LIN {X 0,Y 312.179,Z 630.649,A -85,B 0,C 180,E1 -16129.736,E2 -16129.736} C_VEL
LIN {X 0,Y 313.469,Z 619.934,A -85,B 0,C 180,E1 -16130.85,E2 -16130.85} C_VEL
LIN {X 0,Y 314.719,Z 608.145,A -85,B 0,C 180,E1 -16131.793,E2 -16131.793} C_VEL
LIN {X 0,Y 315.564,Z 595.146,A -85,B 0,C 180,E1 -16132.55,E2 -16132.55} C_VEL
LIN {X 0,Y 316.237,Z 582.572,A -85,B 0,C 180,E1 -16133.017,E2 -16133.017} C_VEL
LIN {X 0,Y 318.093,Z 505.284,A -85,B 0,C 180,E1 -16134.77,E2 -16134.77} C_VEL
LIN {X 0,Y 316.099,Z 493.068,A -85,B 0,C 180,E1 -16135.239,E2 -16135.239} C_VEL
LIN {X 0,Y 314.838,Z 489.465,A -85,B 0,C 180,E1 -16135.437,E2 -16135.437} C_VEL
LIN {X 0,Y 311.272,Z 484.306,A -85,B 0,C 180,E1 -16135.88,E2 -16135.88} C_VEL
LIN {X 0,Y 307.616,Z 479.185,A -85,B 0,C 180,E1 -16136.343,E2 -16136.343} C_VEL
LIN {X 0,Y 306.216,Z 475.627,A -85,B 0,C 180,E1 -16136.565,E2 -16136.565} C_VEL
LIN {X 0,Y 305.882,Z 473.673,A -85,B 0,C 180,E1 -16136.672,E2 -16136.672} C_VEL
LIN {X 0,Y 306.215,Z 468.394,A -85,B 0,C 180,E1 -16137.691,E2 -16137.691} C_VEL
LIN {X 0,Y 304.061,Z 457.591,A -85,B 0,C 180,E1 -16140.18,E2 -16140.18} C_VEL
LIN {X 0,Y 301.282,Z 446.622,A -85,B 0,C 180,E1 -16142.883,E2 -16142.883} C_VEL
LIN {X 0,Y 298.434,Z 436.313,A -85,B 0,C 180,E1 -16145.617,E2 -16145.617} C_VEL
LIN {X 0,Y 298.405,Z 436.31,A -85,B 0,C 180,E1 -16149.487,E2 -16149.487} C_VEL
LIN {X 0,Y 298.428,Z 436.305,A -85,B 0,C 180,E1 -16153.109,E2 -16153.109} C_VEL
LIN {X 0,Y 298.405,Z 436.311,A -85,B 0,C 180,E1 -16156.921,E2 -16156.921} C_VEL
LIN {X 0,Y 298.417,Z 436.315,A -85,B 0,C 180,E1 -16161.004,E2 -16161.004} C_VEL
LIN {X 0,Y 298.42,Z 436.293,A -85,B 0,C 180,E1 -16163.93,E2 -16163.93} C_VEL
LIN {X 0,Y 298.474,Z 436.324,A -85,B 0,C 180,E1 -16168.22,E2 -16168.22} C_VEL
LIN {X 0,Y 302.26,Z 454.228,A -85,B 0,C 180,E1 -16172.288,E2 -16172.288} C_VEL
LIN {X 0,Y 303.264,Z 459.72,A -85,B 0,C 180,E1 -16173.505,E2 -16173.505} C_VEL
LIN {X 0,Y 302.676,Z 470.14,A -85,B 0,C 180,E1 -16175.66,E2 -16175.66} C_VEL
LIN {X 0,Y 302.344,Z 474.693,A -85,B 0,C 180,E1 -16176.542,E2 -16176.542} C_VEL
LIN {X 0,Y 305.64,Z 502.289,A -85,B 0,C 180,E1 -16177.661,E2 -16177.661} C_VEL
LIN {X 0,Y 304.094,Z 552.285,A -85,B 0,C 180,E1 -16179.363,E2 -16179.363} C_VEL
LIN {X 0,Y 302.929,Z 586.5,A -85,B 0,C 180,E1 -16180.562,E2 -16180.562} C_VEL
LIN {X 0,Y 302.336,Z 599.637,A -85,B 0,C 180,E1 -16181.272,E2 -16181.272} C_VEL
LIN {X 0,Y 301.515,Z 612.031,A -85,B 0,C 180,E1 -16182.186,E2 -16182.186} C_VEL
LIN {X 0,Y 300.641,Z 624.863,A -85,B 0,C 180,E1 -16183.426,E2 -16183.426} C_VEL
LIN {X 0,Y 299.793,Z 636.649,A -85,B 0,C 180,E1 -16184.882,E2 -16184.882} C_VEL
LIN {X 0,Y 298.982,Z 646.67,A -85,B 0,C 180,E1 -16186.404,E2 -16186.404} C_VEL
LIN {X 0,Y 298.186,Z 655.778,A -85,B 0,C 180,E1 -16188.098,E2 -16188.098} C_VEL
LIN {X 0,Y 297.536,Z 664.71,A -85,B 0,C 180,E1 -16190.139,E2 -16190.139} C_VEL
LIN {X 0,Y 297.038,Z 671.83,A -85,B 0,C 180,E1 -16192.181,E2 -16192.181} C_VEL
LIN {X 0,Y 296.739,Z 677.24,A -85,B 0,C 180,E1 -16194.119,E2 -16194.119} C_VEL
LIN {X 0,Y 296.671,Z 681.217,A -85,B 0,C 180,E1 -16195.925,E2 -16195.925} C_VEL
LIN {X 0,Y 296.593,Z 683.617,A -85,B 0,C 180,E1 -16197.284,E2 -16197.284} C_VEL
LIN {X 0,Y 296.5,Z 685.517,A -85,B 0,C 180,E1 -16198.642,E2 -16198.642} C_VEL
LIN {X 0,Y 296.504,Z 686.947,A -85,B 0,C 180,E1 -16200,E2 -16200} C_VEL
LIN {X 0,Y 296.551,Z 687.964,A -85,B 0,C 180,E1 -16201.358,E2 -16201.358} C_VEL
LIN {X 0,Y 296.657,Z 688.505,A -85,B 0,C 180,E1 -16202.716,E2 -16202.716} C_VEL
LIN {X 0,Y 296.84,Z 688.612,A -85,B 0,C 180,E1 -16204.073,E2 -16204.073} C_VEL
LIN {X 0,Y 297.108,Z 688.306,A -85,B 0,C 180,E1 -16205.429,E2 -16205.429} C_VEL
LIN {X 0,Y 297.541,Z 687.205,A -85,B 0,C 180,E1 -16207.228,E2 -16207.228} C_VEL
LIN {X 0,Y 298.367,Z 684.756,A -85,B 0,C 180,E1 -16209.49,E2 -16209.49} C_VEL
LIN {X 0,Y 299.443,Z 681.451,A -85,B 0,C 180,E1 -16211.508,E2 -16211.508} C_VEL
LIN {X 0,Y 300.726,Z 677.059,A -85,B 0,C 180,E1 -16213.515,E2 -16213.515} C_VEL
LIN {X 0,Y 302.84,Z 670.363,A -85,B 0,C 180,E1 -16215.824,E2 -16215.824} C_VEL
LIN {X 0,Y 304.885,Z 663.119,A -85,B 0,C 180,E1 -16217.784,E2 -16217.784} C_VEL
LIN {X 0,Y 307.4,Z 654.112,A -85,B 0,C 180,E1 -16219.708,E2 -16219.708} C_VEL
LIN {X 0,Y 310.013,Z 643.808,A -85,B 0,C 180,E1 -16221.477,E2 -16221.477} C_VEL
LIN {X 0,Y 312.558,Z 632.651,A -85,B 0,C 180,E1 -16222.997,E2 -16222.997} C_VEL
LIN {X 0,Y 315.097,Z 619.91,A -85,B 0,C 180,E1 -16224.37,E2 -16224.37} C_VEL
LIN {X 0,Y 317.22,Z 607.363,A -85,B 0,C 180,E1 -16225.42,E2 -16225.42} C_VEL
LIN {X 0,Y 319.135,Z 593.779,A -85,B 0,C 180,E1 -16226.264,E2 -16226.264} C_VEL
LIN {X 0,Y 321.132,Z 574.897,A -85,B 0,C 180,E1 -16227.052,E2 -16227.052} C_VEL
LIN {X 0,Y 327.681,Z 513.253,A -85,B 0,C 180,E1 -16229.483,E2 -16229.483} C_VEL
LIN {X 0,Y 326.096,Z 500.284,A -85,B 0,C 180,E1 -16230.744,E2 -16230.744} C_VEL
LIN {X 0,Y 324.925,Z 493.87,A -85,B 0,C 180,E1 -16231.522,E2 -16231.522} C_VEL
LIN {X 0,Y 322.191,Z 487.566,A -85,B 0,C 180,E1 -16232.816,E2 -16232.816} C_VEL
LIN {X 0,Y 319.761,Z 482.587,A -85,B 0,C 180,E1 -16234.074,E2 -16234.074} C_VEL
LIN {X 0,Y 317.79,Z 478.528,A -85,B 0,C 180,E1 -16235.296,E2 -16235.296} C_VEL
LIN {X 0,Y 316.946,Z 473.742,A -85,B 0,C 180,E1 -16237.86,E2 -16237.86} C_VEL
LIN {X 0,Y 316.18,Z 470.661,A -85,B 0,C 180,E1 -16240.136,E2 -16240.136} C_VEL
LIN {X 0,Y 315.657,Z 468.393,A -85,B 0,C 180,E1 -16242.715,E2 -16242.715} C_VEL
LIN {X 0,Y 315.648,Z 467.284,A -85,B 0,C 180,E1 -16245.438,E2 -16245.438} C_VEL
LIN {X 0,Y 316.37,Z 467.578,A -85,B 0,C 180,E1 -16248.207,E2 -16248.207} C_VEL
LIN {X 0,Y 317.787,Z 469.248,A -85,B 0,C 180,E1 -16250.718,E2 -16250.718} C_VEL
LIN {X 0,Y 319.247,Z 471,A -85,B 0,C 180,E1 -16252.421,E2 -16252.421} C_VEL
LIN {X 0,Y 321.45,Z 475.13,A -85,B 0,C 180,E1 -16254.702,E2 -16254.702} C_VEL
LIN {X 0,Y 322.031,Z 482.327,A -85,B 0,C 180,E1 -16256.56,E2 -16256.56} C_VEL
LIN {X 0,Y 322.94,Z 486.125,A -85,B 0,C 180,E1 -16257.187,E2 -16257.187} C_VEL
LIN {X 0,Y 324.106,Z 499.658,A -85,B 0,C 180,E1 -16258.612,E2 -16258.612} C_VEL
LIN {X 0,Y 324.959,Z 512.771,A -85,B 0,C 180,E1 -16259.773,E2 -16259.773} C_VEL
LIN {X 0,Y 325.209,Z 525.188,A -85,B 0,C 180,E1 -16260.675,E2 -16260.675} C_VEL
LIN {X 0,Y 324.849,Z 536.213,A -85,B 0,C 180,E1 -16261.317,E2 -16261.317} C_VEL
LIN {X 0,Y 317.393,Z 605.626,A -85,B 0,C 180,E1 -16264.111,E2 -16264.111} C_VEL
LIN {X 0,Y 315.334,Z 619.995,A -85,B 0,C 180,E1 -16264.947,E2 -16264.947} C_VEL
LIN {X 0,Y 313.027,Z 633.136,A -85,B 0,C 180,E1 -16265.987,E2 -16265.987} C_VEL
LIN {X 0,Y 310.315,Z 646.166,A -85,B 0,C 180,E1 -16267.355,E2 -16267.355} C_VEL
LIN {X 0,Y 307.955,Z 656.683,A -85,B 0,C 180,E1 -16268.759,E2 -16268.759} C_VEL
LIN {X 0,Y 305.816,Z 665.619,A -85,B 0,C 180,E1 -16270.221,E2 -16270.221} C_VEL
LIN {X 0,Y 303.454,Z 674.922,A -85,B 0,C 180,E1 -16272.091,E2 -16272.091} C_VEL
LIN {X 0,Y 301.362,Z 682.883,A -85,B 0,C 180,E1 -16274.096,E2 -16274.096} C_VEL
LIN {X 0,Y 300.01,Z 688.24,A -85,B 0,C 180,E1 -16275.761,E2 -16275.761} C_VEL
LIN {X 0,Y 298.681,Z 693.437,A -85,B 0,C 180,E1 -16277.774,E2 -16277.774} C_VEL
LIN {X 0,Y 297.725,Z 697.491,A -85,B 0,C 180,E1 -16279.802,E2 -16279.802} C_VEL
LIN {X 0,Y 297.065,Z 700.459,A -85,B 0,C 180,E1 -16281.839,E2 -16281.839} C_VEL
LIN {X 0,Y 296.631,Z 702.706,A -85,B 0,C 180,E1 -16284.324,E2 -16284.324} C_VEL
LIN {X 0,Y 296.602,Z 703.351,A -85,B 0,C 180,E1 -16285.924,E2 -16285.924} C_VEL
LIN {X 0,Y 296.578,Z 703.936,A -85,B 0,C 180,E1 -16290,E2 -16290} C_VEL
LIN {X 0,Y 296.539,Z 703.71,A -85,B 0,C 180,E1 -16291.358,E2 -16291.358} C_VEL
LIN {X 0,Y 296.581,Z 703.091,A -85,B 0,C 180,E1 -16292.716,E2 -16292.716} C_VEL
LIN {X 0,Y 296.576,Z 702.079,A -85,B 0,C 180,E1 -16294.077,E2 -16294.077} C_VEL
LIN {X 0,Y 296.606,Z 700.394,A -85,B 0,C 180,E1 -16295.626,E2 -16295.626} C_VEL
LIN {X 0,Y 296.954,Z 696.415,A -85,B 0,C 180,E1 -16298.164,E2 -16298.164} C_VEL
LIN {X 0,Y 297.44,Z 691.994,A -85,B 0,C 180,E1 -16300.207,E2 -16300.207} C_VEL
LIN {X 0,Y 298.388,Z 685.265,A -85,B 0,C 180,E1 -16302.584,E2 -16302.584} C_VEL
LIN {X 0,Y 299.63,Z 677.919,A -85,B 0,C 180,E1 -16304.605,E2 -16304.605} C_VEL
LIN {X 0,Y 300.821,Z 670.414,A -85,B 0,C 180,E1 -16306.281,E2 -16306.281} C_VEL
LIN {X 0,Y 302.155,Z 661.31,A -85,B 0,C 180,E1 -16307.95,E2 -16307.95} C_VEL
LIN {X 0,Y 303.528,Z 652.857,A -85,B 0,C 180,E1 -16309.266,E2 -16309.266} C_VEL
LIN {X 0,Y 306.344,Z 641.93,A -85,B 0,C 180,E1 -16311.182,E2 -16311.182} C_VEL
LIN {X 0,Y 309.11,Z 630.854,A -85,B 0,C 180,E1 -16312.738,E2 -16312.738} C_VEL
LIN {X 0,Y 311.935,Z 618.673,A -85,B 0,C 180,E1 -16314.102,E2 -16314.102} C_VEL
LIN {X 0,Y 314.837,Z 605.198,A -85,B 0,C 180,E1 -16315.272,E2 -16315.272} C_VEL
LIN {X 0,Y 317.33,Z 591.028,A -85,B 0,C 180,E1 -16316.204,E2 -16316.204} C_VEL
LIN {X 0,Y 319.306,Z 576.399,A -85,B 0,C 180,E1 -16316.91,E2 -16316.91} C_VEL
LIN {X 0,Y 323.506,Z 532.518,A -85,B 0,C 180,E1 -16318.639,E2 -16318.639} C_VEL
LIN {X 0,Y 323.456,Z 521.067,A -85,B 0,C 180,E1 -16319.348,E2 -16319.348} C_VEL
LIN {X 0,Y 322.626,Z 507.921,A -85,B 0,C 180,E1 -16320.374,E2 -16320.374} C_VEL
LIN {X 0,Y 321.365,Z 496.387,A -85,B 0,C 180,E1 -16321.471,E2 -16321.471} C_VEL
LIN {X 0,Y 319.999,Z 486.16,A -85,B 0,C 180,E1 -16322.596,E2 -16322.596} C_VEL
LIN {X 0,Y 317.791,Z 480.722,A -85,B 0,C 180,E1 -16323.689,E2 -16323.689} C_VEL
LIN {X 0,Y 314.86,Z 474.071,A -85,B 0,C 180,E1 -16325.29,E2 -16325.29} C_VEL
LIN {X 0,Y 310.76,Z 465.64,A -85,B 0,C 180,E1 -16328.018,E2 -16328.018} C_VEL
LIN {X 0,Y 307.898,Z 460.525,A -85,B 0,C 180,E1 -16330.617,E2 -16330.617} C_VEL
LIN {X 0,Y 306.358,Z 457.152,A -85,B 0,C 180,E1 -16333.019,E2 -16333.019} C_VEL
LIN {X 0,Y 305.84,Z 455.139,A -85,B 0,C 180,E1 -16335.427,E2 -16335.427} C_VEL
LIN {X 0,Y 306.109,Z 454.482,A -85,B 0,C 180,E1 -16337.282,E2 -16337.282} C_VEL
LIN {X 0,Y 307.974,Z 454.466,A -85,B 0,C 180,E1 -16340.285,E2 -16340.285} C_VEL
LIN {X 0,Y 310.912,Z 457.042,A -85,B 0,C 180,E1 -16343.023,E2 -16343.023} C_VEL
LIN {X 0,Y 311.867,Z 458.038,A -85,B 0,C 180,E1 -16343.717,E2 -16343.717} C_VEL
LIN {X 0,Y 315.045,Z 461.304,A -85,B 0,C 180,E1 -16345.629,E2 -16345.629} C_VEL
LIN {X 0,Y 318.095,Z 465.04,A -85,B 0,C 180,E1 -16347.173,E2 -16347.173} C_VEL
LIN {X 0,Y 321.283,Z 469.175,A -85,B 0,C 180,E1 -16348.553,E2 -16348.553} C_VEL
LIN {X 0,Y 325.804,Z 475.942,A -85,B 0,C 180,E1 -16350.309,E2 -16350.309} C_VEL
LIN {X 0,Y 327.91,Z 479.942,A -85,B 0,C 180,E1 -16351.098,E2 -16351.098} C_VEL
LIN {X 0,Y 321.93,Z 534.652,A -85,B 0,C 180,E1 -16353.283,E2 -16353.283} C_VEL
LIN {X 0,Y 320.518,Z 549.088,A -85,B 0,C 180,E1 -16354.028,E2 -16354.028} C_VEL
LIN {X 0,Y 319.036,Z 561.414,A -85,B 0,C 180,E1 -16354.908,E2 -16354.908} C_VEL
LIN {X 0,Y 316.909,Z 574.47,A -85,B 0,C 180,E1 -16356.124,E2 -16356.124} C_VEL
LIN {X 0,Y 314.538,Z 586.079,A -85,B 0,C 180,E1 -16357.503,E2 -16357.503} C_VEL
LIN {X 0,Y 312.356,Z 595.61,A -85,B 0,C 180,E1 -16358.9,E2 -16358.9} C_VEL
LIN {X 0,Y 310.19,Z 604.328,A -85,B 0,C 180,E1 -16360.477,E2 -16360.477} C_VEL
LIN {X 0,Y 308.126,Z 611.561,A -85,B 0,C 180,E1 -16362.066,E2 -16362.066} C_VEL
LIN {X 0,Y 305.926,Z 618.701,A -85,B 0,C 180,E1 -16363.998,E2 -16363.998} C_VEL
LIN {X 0,Y 303.95,Z 624.421,A -85,B 0,C 180,E1 -16365.949,E2 -16365.949} C_VEL
LIN {X 0,Y 302.306,Z 628.869,A -85,B 0,C 180,E1 -16367.923,E2 -16367.923} C_VEL
LIN {X 0,Y 301.275,Z 631.244,A -85,B 0,C 180,E1 -16369.244,E2 -16369.244} C_VEL
LIN {X 0,Y 300.367,Z 633.147,A -85,B 0,C 180,E1 -16370.573,E2 -16370.573} C_VEL
LIN {X 0,Y 299.648,Z 634.568,A -85,B 0,C 180,E1 -16371.91,E2 -16371.91} C_VEL
LIN {X 0,Y 299.074,Z 635.563,A -85,B 0,C 180,E1 -16373.252,E2 -16373.252} C_VEL
LIN {X 0,Y 298.54,Z 636.139,A -85,B 0,C 180,E1 -16374.597,E2 -16374.597} C_VEL
LIN {X 0,Y 298.063,Z 636.261,A -85,B 0,C 180,E1 -16375.944,E2 -16375.944} C_VEL
LIN {X 0,Y 297.707,Z 635.969,A -85,B 0,C 180,E1 -16377.294,E2 -16377.294} C_VEL
LIN {X 0,Y 297.453,Z 635.269,A -85,B 0,C 180,E1 -16378.646,E2 -16378.646} C_VEL
LIN {X 0,Y 297.297,Z 634.103,A -85,B 0,C 180,E1 -16380,E2 -16380} C_VEL
LIN {X 0,Y 297.313,Z 631.537,A -85,B 0,C 180,E1 -16382.032,E2 -16382.032} C_VEL
LIN {X 0,Y 297.458,Z 627.933,A -85,B 0,C 180,E1 -16384.065,E2 -16384.065} C_VEL
LIN {X 0,Y 297.67,Z 623.195,A -85,B 0,C 180,E1 -16386.099,E2 -16386.099} C_VEL
LIN {X 0,Y 298.012,Z 616.074,A -85,B 0,C 180,E1 -16388.476,E2 -16388.476} C_VEL
LIN {X 0,Y 298.523,Z 608.297,A -85,B 0,C 180,E1 -16390.513,E2 -16390.513} C_VEL
LIN {X 0,Y 299.307,Z 598.647,A -85,B 0,C 180,E1 -16392.545,E2 -16392.545} C_VEL
LIN {X 0,Y 300.184,Z 587.588,A -85,B 0,C 180,E1 -16394.404,E2 -16394.404} C_VEL
LIN {X 0,Y 300.941,Z 576.409,A -85,B 0,C 180,E1 -16395.927,E2 -16395.927} C_VEL
LIN {X 0,Y 301.806,Z 564.264,A -85,B 0,C 180,E1 -16397.239,E2 -16397.239} C_VEL
LIN {X 0,Y 302.449,Z 550.933,A -85,B 0,C 180,E1 -16398.37,E2 -16398.37} C_VEL
LIN {X 0,Y 303.109,Z 536.628,A -85,B 0,C 180,E1 -16399.25,E2 -16399.25} C_VEL
LIN {X 0,Y 303.479,Z 522.328,A -85,B 0,C 180,E1 -16399.841,E2 -16399.841} C_VEL
LIN {X 0,Y 305.469,Z 458.71,A -85,B 0,C 180,E1 -16402.009,E2 -16402.009} C_VEL
LIN {X 0,Y 298.462,Z 436.299,A -85,B 0,C 180,E1 -16403.13,E2 -16403.13} C_VEL
LIN {X 0,Y 298.486,Z 436.303,A -85,B 0,C 180,E1 -16406.575,E2 -16406.575} C_VEL
LIN {X 0,Y 298.419,Z 436.314,A -85,B 0,C 180,E1 -16409.641,E2 -16409.641} C_VEL
LIN {X 0,Y 298.397,Z 436.29,A -85,B 0,C 180,E1 -16412.8,E2 -16412.8} C_VEL
LIN {X 0,Y 298.449,Z 436.311,A -85,B 0,C 180,E1 -16416.808,E2 -16416.808} C_VEL
LIN {X 0,Y 298.411,Z 436.3,A -85,B 0,C 180,E1 -16419.486,E2 -16419.486} C_VEL
LIN {X 0,Y 298.4,Z 436.321,A -85,B 0,C 180,E1 -16423.103,E2 -16423.103} C_VEL
LIN {X 0,Y 298.405,Z 436.305,A -85,B 0,C 180,E1 -16426.921,E2 -16426.921} C_VEL
LIN {X 0,Y 298.417,Z 436.309,A -85,B 0,C 180,E1 -16431.004,E2 -16431.004} C_VEL
LIN {X 0,Y 298.429,Z 436.362,A -85,B 0,C 180,E1 -16434.547,E2 -16434.547} C_VEL
LIN {X 0,Y 301.7,Z 448.047,A -85,B 0,C 180,E1 -16437.603,E2 -16437.603} C_VEL
LIN {X 0,Y 304.671,Z 460.525,A -85,B 0,C 180,E1 -16440.647,E2 -16440.647} C_VEL
LIN {X 0,Y 306.128,Z 467.823,A -85,B 0,C 180,E1 -16442.314,E2 -16442.314} C_VEL
LIN {X 0,Y 305.847,Z 473.764,A -85,B 0,C 180,E1 -16443.462,E2 -16443.462} C_VEL
LIN {X 0,Y 310.58,Z 499.528,A -85,B 0,C 180,E1 -16444.558,E2 -16444.558} C_VEL
LIN {X 0,Y 311.587,Z 506.235,A -85,B 0,C 180,E1 -16444.814,E2 -16444.814} C_VEL
LIN {X 0,Y 309.769,Z 580.357,A -85,B 0,C 180,E1 -16446.518,E2 -16446.518} C_VEL
LIN {X 0,Y 309.181,Z 593.095,A -85,B 0,C 180,E1 -16446.958,E2 -16446.958} C_VEL
LIN {X 0,Y 308.244,Z 605.504,A -85,B 0,C 180,E1 -16447.637,E2 -16447.637} C_VEL
LIN {X 0,Y 307.165,Z 617.161,A -85,B 0,C 180,E1 -16448.526,E2 -16448.526} C_VEL
LIN {X 0,Y 305.785,Z 628.549,A -85,B 0,C 180,E1 -16449.658,E2 -16449.658} C_VEL
LIN {X 0,Y 304.37,Z 638.81,A -85,B 0,C 180,E1 -16450.965,E2 -16450.965} C_VEL
LIN {X 0,Y 303.085,Z 648.214,A -85,B 0,C 180,E1 -16452.455,E2 -16452.455} C_VEL
LIN {X 0,Y 301.533,Z 656.811,A -85,B 0,C 180,E1 -16454.106,E2 -16454.106} C_VEL
LIN {X 0,Y 300.238,Z 663.905,A -85,B 0,C 180,E1 -16455.772,E2 -16455.772} C_VEL
LIN {X 0,Y 299.08,Z 670.867,A -85,B 0,C 180,E1 -16457.79,E2 -16457.79} C_VEL
LIN {X 0,Y 298.096,Z 676.399,A -85,B 0,C 180,E1 -16459.815,E2 -16459.815} C_VEL
LIN {X 0,Y 297.441,Z 680.736,A -85,B 0,C 180,E1 -16461.85,E2 -16461.85} C_VEL
LIN {X 0,Y 297.107,Z 683.412,A -85,B 0,C 180,E1 -16463.467,E2 -16463.467} C_VEL
LIN {X 0,Y 296.766,Z 686.296,A -85,B 0,C 180,E1 -16465.926,E2 -16465.926} C_VEL
LIN {X 0,Y 296.53,Z 687.905,A -85,B 0,C 180,E1 -16468.642,E2 -16468.642} C_VEL
LIN {X 0,Y 296.512,Z 688.138,A -85,B 0,C 180,E1 -16470,E2 -16470} C_VEL
LIN {X 0,Y 296.53,Z 687.944,A -85,B 0,C 180,E1 -16471.358,E2 -16471.358} C_VEL
LIN {X 0,Y 296.765,Z 686.385,A -85,B 0,C 180,E1 -16474.074,E2 -16474.074} C_VEL
LIN {X 0,Y 297.076,Z 683.66,A -85,B 0,C 180,E1 -16476.482,E2 -16476.482} C_VEL
LIN {X 0,Y 297.608,Z 679.632,A -85,B 0,C 180,E1 -16478.83,E2 -16478.83} C_VEL
LIN {X 0,Y 298.379,Z 674.966,A -85,B 0,C 180,E1 -16480.861,E2 -16480.861} C_VEL
LIN {X 0,Y 299.636,Z 667.955,A -85,B 0,C 180,E1 -16483.22,E2 -16483.22} C_VEL
LIN {X 0,Y 300.963,Z 660.269,A -85,B 0,C 180,E1 -16485.231,E2 -16485.231} C_VEL
LIN {X 0,Y 302.672,Z 650.694,A -85,B 0,C 180,E1 -16487.221,E2 -16487.221} C_VEL
LIN {X 0,Y 304.1,Z 640.694,A -85,B 0,C 180,E1 -16488.878,E2 -16488.878} C_VEL
LIN {X 0,Y 305.753,Z 629.442,A -85,B 0,C 180,E1 -16490.344,E2 -16490.344} C_VEL
LIN {X 0,Y 307.069,Z 618.385,A -85,B 0,C 180,E1 -16491.481,E2 -16491.481} C_VEL
LIN {X 0,Y 308.323,Z 605.869,A -85,B 0,C 180,E1 -16492.446,E2 -16492.446} C_VEL
LIN {X 0,Y 309.196,Z 592.749,A -85,B 0,C 180,E1 -16493.173,E2 -16493.173} C_VEL
LIN {X 0,Y 309.847,Z 579.653,A -85,B 0,C 180,E1 -16493.608,E2 -16493.608} C_VEL
LIN {X 0,Y 311.632,Z 505.741,A -85,B 0,C 180,E1 -16495.309,E2 -16495.309} C_VEL
LIN {X 0,Y 306.363,Z 476.274,A -85,B 0,C 180,E1 -16496.534,E2 -16496.534} C_VEL
LIN {X 0,Y 306.216,Z 475.627,A -85,B 0,C 180,E1 -16496.565,E2 -16496.565} C_VEL
LIN {X 0,Y 305.484,Z 473.734,A -85,B 0,C 180,E1 -16496.76,E2 -16496.76} C_VEL
LIN {X 0,Y 301.109,Z 467.447,A -85,B 0,C 180,E1 -16498.408,E2 -16498.408} C_VEL
LIN {X 0,Y 298.495,Z 462.57,A -85,B 0,C 180,E1 -16499.778,E2 -16499.778} C_VEL
LIN {X 0,Y 296.804,Z 457.027,A -85,B 0,C 180,E1 -16501.125,E2 -16501.125} C_VEL
LIN {X 0,Y 293.533,Z 444.563,A -85,B 0,C 180,E1 -16504.308,E2 -16504.308} C_VEL
LIN {X 0,Y 291.384,Z 437.193,A -85,B 0,C 180,E1 -16506.329,E2 -16506.329} C_VEL
LIN {X 0,Y 291.351,Z 437.186,A -85,B 0,C 180,E1 -16510.64,E2 -16510.64} C_VEL
LIN {X 0,Y 291.324,Z 437.189,A -85,B 0,C 180,E1 -16514.396,E2 -16514.396} C_VEL
LIN {X 0,Y 291.329,Z 437.183,A -85,B 0,C 180,E1 -16518.404,E2 -16518.404} C_VEL
LIN {X 0,Y 291.366,Z 437.192,A -85,B 0,C 180,E1 -16521.16,E2 -16521.16} C_VEL
LIN {X 0,Y 291.363,Z 437.177,A -85,B 0,C 180,E1 -16524.626,E2 -16524.626} C_VEL
LIN {X 0,Y 291.405,Z 437.319,A -85,B 0,C 180,E1 -16527.955,E2 -16527.955} C_VEL
LIN {X 0,Y 294.986,Z 454.043,A -85,B 0,C 180,E1 -16531.827,E2 -16531.827} C_VEL
LIN {X 0,Y 296.312,Z 461.968,A -85,B 0,C 180,E1 -16533.597,E2 -16533.597} C_VEL
LIN {X 0,Y 295.389,Z 474.496,A -85,B 0,C 180,E1 -16536.223,E2 -16536.223} C_VEL
LIN {X 0,Y 298.331,Z 500.617,A -85,B 0,C 180,E1 -16537.318,E2 -16537.318} C_VEL
LIN {X 0,Y 298.746,Z 505.394,A -85,B 0,C 180,E1 -16537.51,E2 -16537.51} C_VEL
LIN {X 0,Y 295.885,Z 586.649,A -85,B 0,C 180,E1 -16540.397,E2 -16540.397} C_VEL
LIN {X 0,Y 295.263,Z 600.43,A -85,B 0,C 180,E1 -16541.166,E2 -16541.166} C_VEL
LIN {X 0,Y 294.433,Z 612.646,A -85,B 0,C 180,E1 -16542.102,E2 -16542.102} C_VEL
LIN {X 0,Y 293.538,Z 625.414,A -85,B 0,C 180,E1 -16543.373,E2 -16543.373} C_VEL
LIN {X 0,Y 292.786,Z 635.891,A -85,B 0,C 180,E1 -16544.69,E2 -16544.69} C_VEL
LIN {X 0,Y 291.87,Z 647.106,A -85,B 0,C 180,E1 -16546.422,E2 -16546.422} C_VEL
LIN {X 0,Y 291.058,Z 656.151,A -85,B 0,C 180,E1 -16548.156,E2 -16548.156} C_VEL
LIN {X 0,Y 290.416,Z 665.03,A -85,B 0,C 180,E1 -16550.247,E2 -16550.247} C_VEL
LIN {X 0,Y 289.912,Z 672.102,A -85,B 0,C 180,E1 -16552.338,E2 -16552.338} C_VEL
LIN {X 0,Y 289.626,Z 677.742,A -85,B 0,C 180,E1 -16554.43,E2 -16554.43} C_VEL
LIN {X 0,Y 289.553,Z 682.123,A -85,B 0,C 180,E1 -16556.521,E2 -16556.521} C_VEL
LIN {X 0,Y 289.423,Z 685.345,A -85,B 0,C 180,E1 -16558.608,E2 -16558.608} C_VEL
LIN {X 0,Y 289.423,Z 686.886,A -85,B 0,C 180,E1 -16560,E2 -16560} C_VEL
LIN {X 0,Y 289.472,Z 687.984,A -85,B 0,C 180,E1 -16561.391,E2 -16561.391} C_VEL
LIN {X 0,Y 289.588,Z 688.66,A -85,B 0,C 180,E1 -16562.782,E2 -16562.782} C_VEL
LIN {X 0,Y 289.765,Z 688.869,A -85,B 0,C 180,E1 -16564.173,E2 -16564.173} C_VEL
LIN {X 0,Y 290.054,Z 688.651,A -85,B 0,C 180,E1 -16565.562,E2 -16565.562} C_VEL
LIN {X 0,Y 290.479,Z 687.821,A -85,B 0,C 180,E1 -16567.262,E2 -16567.262} C_VEL
LIN {X 0,Y 291.403,Z 685.424,A -85,B 0,C 180,E1 -16569.719,E2 -16569.719} C_VEL
LIN {X 0,Y 292.553,Z 682.334,A -85,B 0,C 180,E1 -16571.782,E2 -16571.782} C_VEL
LIN {X 0,Y 293.912,Z 678.169,A -85,B 0,C 180,E1 -16573.835,E2 -16573.835} C_VEL
LIN {X 0,Y 296.144,Z 671.733,A -85,B 0,C 180,E1 -16576.191,E2 -16576.191} C_VEL
LIN {X 0,Y 298.344,Z 664.815,A -85,B 0,C 180,E1 -16578.187,E2 -16578.187} C_VEL
LIN {X 0,Y 300.967,Z 656.23,A -85,B 0,C 180,E1 -16580.147,E2 -16580.147} C_VEL
LIN {X 0,Y 303.855,Z 645.783,A -85,B 0,C 180,E1 -16582.036,E2 -16582.036} C_VEL
LIN {X 0,Y 306.542,Z 635.123,A -85,B 0,C 180,E1 -16583.583,E2 -16583.583} C_VEL
LIN {X 0,Y 309.043,Z 623.947,A -85,B 0,C 180,E1 -16584.88,E2 -16584.88} C_VEL
LIN {X 0,Y 311.562,Z 610.511,A -85,B 0,C 180,E1 -16586.095,E2 -16586.095} C_VEL
LIN {X 0,Y 313.63,Z 597.549,A -85,B 0,C 180,E1 -16586.986,E2 -16586.986} C_VEL
LIN {X 0,Y 315.482,Z 583.31,A -85,B 0,C 180,E1 -16587.667,E2 -16587.667} C_VEL
LIN {X 0,Y 323.249,Z 515.302,A -85,B 0,C 180,E1 -16590.4,E2 -16590.4} C_VEL
LIN {X 0,Y 321.95,Z 503.161,A -85,B 0,C 180,E1 -16591.641,E2 -16591.641} C_VEL
LIN {X 0,Y 321.113,Z 498.234,A -85,B 0,C 180,E1 -16592.26,E2 -16592.26} C_VEL
LIN {X 0,Y 318.722,Z 492.519,A -85,B 0,C 180,E1 -16593.514,E2 -16593.514} C_VEL
LIN {X 0,Y 316.917,Z 488.535,A -85,B 0,C 180,E1 -16594.55,E2 -16594.55} C_VEL
LIN {X 0,Y 314.499,Z 483.702,A -85,B 0,C 180,E1 -16596.085,E2 -16596.085} C_VEL
LIN {X 0,Y 312.24,Z 479.103,A -85,B 0,C 180,E1 -16597.946,E2 -16597.946} C_VEL
LIN {X 0,Y 311.56,Z 475.527,A -85,B 0,C 180,E1 -16600.857,E2 -16600.857} C_VEL
LIN {X 0,Y 311.368,Z 474.108,A -85,B 0,C 180,E1 -16602.621,E2 -16602.621} C_VEL
LIN {X 0,Y 311.552,Z 473.018,A -85,B 0,C 180,E1 -16605.629,E2 -16605.629} C_VEL
LIN {X 0,Y 312.254,Z 473.328,A -85,B 0,C 180,E1 -16607.966,E2 -16607.966} C_VEL
LIN {X 0,Y 313.158,Z 474.351,A -85,B 0,C 180,E1 -16609.733,E2 -16609.733} C_VEL
LIN {X 0,Y 315.146,Z 476.68,A -85,B 0,C 180,E1 -16612.173,E2 -16612.173} C_VEL
LIN {X 0,Y 317.213,Z 480.758,A -85,B 0,C 180,E1 -16614.435,E2 -16614.435} C_VEL
LIN {X 0,Y 317.554,Z 483.199,A -85,B 0,C 180,E1 -16615.035,E2 -16615.035} C_VEL
LIN {X 0,Y 319.298,Z 489.713,A -85,B 0,C 180,E1 -16616.315,E2 -16616.315} C_VEL
LIN {X 0,Y 320.288,Z 504.611,A -85,B 0,C 180,E1 -16617.92,E2 -16617.92} C_VEL
LIN {X 0,Y 320.789,Z 519.571,A -85,B 0,C 180,E1 -16619.21,E2 -16619.21} C_VEL
LIN {X 0,Y 320.65,Z 529.629,A -85,B 0,C 180,E1 -16619.911,E2 -16619.911} C_VEL
LIN {X 0,Y 320.261,Z 537.293,A -85,B 0,C 180,E1 -16620.37,E2 -16620.37} C_VEL
LIN {X 0,Y 312.222,Z 606.638,A -85,B 0,C 180,E1 -16623.244,E2 -16623.244} C_VEL
LIN {X 0,Y 310.152,Z 619.948,A -85,B 0,C 180,E1 -16624.048,E2 -16624.048} C_VEL
LIN {X 0,Y 307.835,Z 632.005,A -85,B 0,C 180,E1 -16625.016,E2 -16625.016} C_VEL
LIN {X 0,Y 304.925,Z 645.161,A -85,B 0,C 180,E1 -16626.393,E2 -16626.393} C_VEL
LIN {X 0,Y 302.345,Z 655.795,A -85,B 0,C 180,E1 -16627.807,E2 -16627.807} C_VEL
LIN {X 0,Y 299.528,Z 666.492,A -85,B 0,C 180,E1 -16629.613,E2 -16629.613} C_VEL
LIN {X 0,Y 296.893,Z 676.006,A -85,B 0,C 180,E1 -16631.617,E2 -16631.617} C_VEL
LIN {X 0,Y 294.61,Z 683.879,A -85,B 0,C 180,E1 -16633.722,E2 -16633.722} C_VEL
LIN {X 0,Y 293.179,Z 688.982,A -85,B 0,C 180,E1 -16635.422,E2 -16635.422} C_VEL
LIN {X 0,Y 291.776,Z 693.992,A -85,B 0,C 180,E1 -16637.48,E2 -16637.48} C_VEL
LIN {X 0,Y 290.75,Z 697.83,A -85,B 0,C 180,E1 -16639.555,E2 -16639.555} C_VEL
LIN {X 0,Y 290.041,Z 700.613,A -85,B 0,C 180,E1 -16641.64,E2 -16641.64} C_VEL
LIN {X 0,Y 289.716,Z 701.922,A -85,B 0,C 180,E1 -16643.033,E2 -16643.033} C_VEL
LIN {X 0,Y 289.557,Z 702.757,A -85,B 0,C 180,E1 -16644.429,E2 -16644.429} C_VEL
LIN {X 0,Y 289.503,Z 703.176,A -85,B 0,C 180,E1 -16645.824,E2 -16645.824} C_VEL
LIN {X 0,Y 289.506,Z 703.164,A -85,B 0,C 180,E1 -16647.217,E2 -16647.217} C_VEL
LIN {X 0,Y 289.492,Z 703.748,A -85,B 0,C 180,E1 -16650,E2 -16650} C_VEL
LIN {X 0,Y 289.459,Z 703.521,A -85,B 0,C 180,E1 -16651.391,E2 -16651.391} C_VEL
LIN {X 0,Y 289.506,Z 702.903,A -85,B 0,C 180,E1 -16652.783,E2 -16652.783} C_VEL
LIN {X 0,Y 289.476,Z 701.889,A -85,B 0,C 180,E1 -16654.177,E2 -16654.177} C_VEL
LIN {X 0,Y 289.517,Z 700.451,A -85,B 0,C 180,E1 -16655.572,E2 -16655.572} C_VEL
LIN {X 0,Y 289.743,Z 697.466,A -85,B 0,C 180,E1 -16657.667,E2 -16657.667} C_VEL
LIN {X 0,Y 290.224,Z 693.418,A -85,B 0,C 180,E1 -16659.759,E2 -16659.759} C_VEL
LIN {X 0,Y 291.057,Z 687.177,A -85,B 0,C 180,E1 -16662.198,E2 -16662.198} C_VEL
LIN {X 0,Y 292.261,Z 680.376,A -85,B 0,C 180,E1 -16664.269,E2 -16664.269} C_VEL
LIN {X 0,Y 293.41,Z 673.413,A -85,B 0,C 180,E1 -16665.989,E2 -16665.989} C_VEL
LIN {X 0,Y 294.798,Z 664.983,A -85,B 0,C 180,E1 -16667.699,E2 -16667.699} C_VEL
LIN {X 0,Y 296.26,Z 656.009,A -85,B 0,C 180,E1 -16669.217,E2 -16669.217} C_VEL
LIN {X 0,Y 298.816,Z 646.985,A -85,B 0,C 180,E1 -16671.019,E2 -16671.019} C_VEL
LIN {X 0,Y 301.815,Z 636.053,A -85,B 0,C 180,E1 -16672.776,E2 -16672.776} C_VEL
LIN {X 0,Y 304.947,Z 624.016,A -85,B 0,C 180,E1 -16674.328,E2 -16674.328} C_VEL
LIN {X 0,Y 307.884,Z 612.097,A -85,B 0,C 180,E1 -16675.522,E2 -16675.522} C_VEL
LIN {X 0,Y 310.544,Z 599.356,A -85,B 0,C 180,E1 -16676.549,E2 -16676.549} C_VEL
LIN {X 0,Y 313.244,Z 583.825,A -85,B 0,C 180,E1 -16677.474,E2 -16677.474} C_VEL
LIN {X 0,Y 315.4,Z 565.795,A -85,B 0,C 180,E1 -16678.239,E2 -16678.239} C_VEL
LIN {X 0,Y 318.718,Z 533.68,A -85,B 0,C 180,E1 -16679.551,E2 -16679.551} C_VEL
LIN {X 0,Y 318.741,Z 521.992,A -85,B 0,C 180,E1 -16680.316,E2 -16680.316} C_VEL
LIN {X 0,Y 318.138,Z 509.971,A -85,B 0,C 180,E1 -16681.3,E2 -16681.3} C_VEL
LIN {X 0,Y 317.095,Z 498.477,A -85,B 0,C 180,E1 -16682.44,E2 -16682.44} C_VEL
LIN {X 0,Y 316.146,Z 490.547,A -85,B 0,C 180,E1 -16683.362,E2 -16683.362} C_VEL
LIN {X 0,Y 314.409,Z 485.966,A -85,B 0,C 180,E1 -16684.315,E2 -16684.315} C_VEL
LIN {X 0,Y 311.808,Z 479.676,A -85,B 0,C 180,E1 -16685.876,E2 -16685.876} C_VEL
LIN {X 0,Y 308.307,Z 471.889,A -85,B 0,C 180,E1 -16688.45,E2 -16688.45} C_VEL
LIN {X 0,Y 305.744,Z 466.95,A -85,B 0,C 180,E1 -16691.035,E2 -16691.035} C_VEL
LIN {X 0,Y 304.536,Z 463.938,A -85,B 0,C 180,E1 -16693.196,E2 -16693.196} C_VEL
LIN {X 0,Y 304.103,Z 461.857,A -85,B 0,C 180,E1 -16695.761,E2 -16695.761} C_VEL
LIN {X 0,Y 304.656,Z 461.277,A -85,B 0,C 180,E1 -16698.011,E2 -16698.011} C_VEL
LIN {X 0,Y 306.234,Z 461.427,A -85,B 0,C 180,E1 -16700.33,E2 -16700.33} C_VEL
LIN {X 0,Y 309.461,Z 464.315,A -85,B 0,C 180,E1 -16703.286,E2 -16703.286} C_VEL
LIN {X 0,Y 312.821,Z 468.059,A -85,B 0,C 180,E1 -16705.448,E2 -16705.448} C_VEL
LIN {X 0,Y 315.372,Z 471.242,A -85,B 0,C 180,E1 -16706.801,E2 -16706.801} C_VEL
LIN {X 0,Y 318.941,Z 476.151,A -85,B 0,C 180,E1 -16708.439,E2 -16708.439} C_VEL
LIN {X 0,Y 322.712,Z 482.32,A -85,B 0,C 180,E1 -16709.997,E2 -16709.997} C_VEL
LIN {X 0,Y 323.275,Z 483.538,A -85,B 0,C 180,E1 -16710.225,E2 -16710.225} C_VEL
LIN {X 0,Y 317.144,Z 535.408,A -85,B 0,C 180,E1 -16712.356,E2 -16712.356} C_VEL
LIN {X 0,Y 315.633,Z 549.908,A -85,B 0,C 180,E1 -16713.11,E2 -16713.11} C_VEL
LIN {X 0,Y 314.051,Z 561.634,A -85,B 0,C 180,E1 -16713.961,E2 -16713.961} C_VEL
LIN {X 0,Y 311.778,Z 574.577,A -85,B 0,C 180,E1 -16715.176,E2 -16715.176} C_VEL
LIN {X 0,Y 309.297,Z 586.379,A -85,B 0,C 180,E1 -16716.569,E2 -16716.569} C_VEL
LIN {X 0,Y 306.685,Z 596.843,A -85,B 0,C 180,E1 -16718.137,E2 -16718.137} C_VEL
LIN {X 0,Y 304.309,Z 605.441,A -85,B 0,C 180,E1 -16719.731,E2 -16719.731} C_VEL
LIN {X 0,Y 301.722,Z 613.92,A -85,B 0,C 180,E1 -16721.672,E2 -16721.672} C_VEL
LIN {X 0,Y 299.375,Z 620.733,A -85,B 0,C 180,E1 -16723.638,E2 -16723.638} C_VEL
LIN {X 0,Y 297.23,Z 626.352,A -85,B 0,C 180,E1 -16725.695,E2 -16725.695} C_VEL
LIN {X 0,Y 295.54,Z 630.449,A -85,B 0,C 180,E1 -16727.642,E2 -16727.642} C_VEL
LIN {X 0,Y 294.447,Z 632.674,A -85,B 0,C 180,E1 -16728.992,E2 -16728.992} C_VEL
LIN {X 0,Y 293.48,Z 634.421,A -85,B 0,C 180,E1 -16730.35,E2 -16730.35} C_VEL
LIN {X 0,Y 292.715,Z 635.727,A -85,B 0,C 180,E1 -16731.717,E2 -16731.717} C_VEL
LIN {X 0,Y 292.099,Z 636.605,A -85,B 0,C 180,E1 -16733.091,E2 -16733.091} C_VEL
LIN {X 0,Y 291.54,Z 637.04,A -85,B 0,C 180,E1 -16734.467,E2 -16734.467} C_VEL
LIN {X 0,Y 291.046,Z 637.068,A -85,B 0,C 180,E1 -16735.846,E2 -16735.846} C_VEL
LIN {X 0,Y 290.677,Z 636.681,A -85,B 0,C 180,E1 -16737.228,E2 -16737.228} C_VEL
LIN {X 0,Y 290.385,Z 635.833,A -85,B 0,C 180,E1 -16738.613,E2 -16738.613} C_VEL
LIN {X 0,Y 290.23,Z 634.558,A -85,B 0,C 180,E1 -16740,E2 -16740} C_VEL
LIN {X 0,Y 290.249,Z 631.826,A -85,B 0,C 180,E1 -16742.082,E2 -16742.082} C_VEL
LIN {X 0,Y 290.377,Z 628.039,A -85,B 0,C 180,E1 -16744.164,E2 -16744.164} C_VEL
LIN {X 0,Y 290.596,Z 623.099,A -85,B 0,C 180,E1 -16746.248,E2 -16746.248} C_VEL
LIN {X 0,Y 290.894,Z 616.869,A -85,B 0,C 180,E1 -16748.335,E2 -16748.335} C_VEL
LIN {X 0,Y 291.399,Z 609.091,A -85,B 0,C 180,E1 -16750.421,E2 -16750.421} C_VEL
LIN {X 0,Y 292.192,Z 599.48,A -85,B 0,C 180,E1 -16752.502,E2 -16752.502} C_VEL
LIN {X 0,Y 293.052,Z 588.489,A -85,B 0,C 180,E1 -16754.407,E2 -16754.407} C_VEL
LIN {X 0,Y 293.815,Z 577.399,A -85,B 0,C 180,E1 -16755.967,E2 -16755.967} C_VEL
LIN {X 0,Y 294.636,Z 565.813,A -85,B 0,C 180,E1 -16757.27,E2 -16757.27} C_VEL
LIN {X 0,Y 295.364,Z 552.214,A -85,B 0,C 180,E1 -16758.467,E2 -16758.467} C_VEL
LIN {X 0,Y 296.057,Z 538.177,A -85,B 0,C 180,E1 -16759.366,E2 -16759.366} C_VEL
LIN {X 0,Y 296.425,Z 524.446,A -85,B 0,C 180,E1 -16759.972,E2 -16759.972} C_VEL
LIN {X 0,Y 298.546,Z 460.094,A -85,B 0,C 180,E1 -16762.231,E2 -16762.231} C_VEL
LIN {X 0,Y 291.413,Z 437.177,A -85,B 0,C 180,E1 -16763.417,E2 -16763.417} C_VEL
LIN {X 0,Y 291.417,Z 437.178,A -85,B 0,C 180,E1 -16767.272,E2 -16767.272} C_VEL
LIN {X 0,Y 291.336,Z 437.194,A -85,B 0,C 180,E1 -16770.437,E2 -16770.437} C_VEL
LIN {X 0,Y 291.346,Z 437.163,A -85,B 0,C 180,E1 -16773.698,E2 -16773.698} C_VEL
LIN {X 0,Y 291.384,Z 437.194,A -85,B 0,C 180,E1 -16777.256,E2 -16777.256} C_VEL
LIN {X 0,Y 291.336,Z 437.176,A -85,B 0,C 180,E1 -16780.642,E2 -16780.642} C_VEL
LIN {X 0,Y 291.292,Z 437.196,A -85,B 0,C 180,E1 -16784.402,E2 -16784.402} C_VEL
LIN {X 0,Y 291.328,Z 437.196,A -85,B 0,C 180,E1 -16788.404,E2 -16788.404} C_VEL
LIN {X 0,Y 291.366,Z 437.189,A -85,B 0,C 180,E1 -16791.16,E2 -16791.16} C_VEL
LIN {X 0,Y 291.42,Z 437.326,A -85,B 0,C 180,E1 -16793.871,E2 -16793.871} C_VEL
LIN {X 0,Y 294.861,Z 449.458,A -85,B 0,C 180,E1 -16797.106,E2 -16797.106} C_VEL
LIN {X 0,Y 297.578,Z 460.615,A -85,B 0,C 180,E1 -16799.894,E2 -16799.894} C_VEL
LIN {X 0,Y 299.422,Z 469.656,A -85,B 0,C 180,E1 -16802.002,E2 -16802.002} C_VEL
LIN {X 0,Y 299.341,Z 474.181,A -85,B 0,C 180,E1 -16802.855,E2 -16802.855} C_VEL
LIN {X 0,Y 304.241,Z 500.909,A -85,B 0,C 180,E1 -16804.022,E2 -16804.022} C_VEL
LIN {X 0,Y 305.168,Z 507.831,A -85,B 0,C 180,E1 -16804.285,E2 -16804.285} C_VEL
LIN {X 0,Y 303.284,Z 580.469,A -85,B 0,C 180,E1 -16805.985,E2 -16805.985} C_VEL
LIN {X 0,Y 302.683,Z 593.248,A -85,B 0,C 180,E1 -16806.434,E2 -16806.434} C_VEL
LIN {X 0,Y 301.691,Z 605.671,A -85,B 0,C 180,E1 -16807.124,E2 -16807.124} C_VEL
LIN {X 0,Y 300.591,Z 617.335,A -85,B 0,C 180,E1 -16808.032,E2 -16808.032} C_VEL
LIN {X 0,Y 299.148,Z 628.728,A -85,B 0,C 180,E1 -16809.186,E2 -16809.186} C_VEL
LIN {X 0,Y 297.482,Z 640.13,A -85,B 0,C 180,E1 -16810.686,E2 -16810.686} C_VEL
LIN {X 0,Y 295.974,Z 650.292,A -85,B 0,C 180,E1 -16812.377,E2 -16812.377} C_VEL
LIN {X 0,Y 294.154,Z 659.986,A -85,B 0,C 180,E1 -16814.408,E2 -16814.408} C_VEL
LIN {X 0,Y 292.76,Z 667.771,A -85,B 0,C 180,E1 -16816.464,E2 -16816.464} C_VEL
LIN {X 0,Y 291.77,Z 673.029,A -85,B 0,C 180,E1 -16818.185,E2 -16818.185} C_VEL
LIN {X 0,Y 290.845,Z 678.165,A -85,B 0,C 180,E1 -16820.262,E2 -16820.262} C_VEL
LIN {X 0,Y 290.247,Z 682.138,A -85,B 0,C 180,E1 -16822.347,E2 -16822.347} C_VEL
LIN {X 0,Y 289.831,Z 685.067,A -85,B 0,C 180,E1 -16824.434,E2 -16824.434} C_VEL
LIN {X 0,Y 289.687,Z 686.485,A -85,B 0,C 180,E1 -16825.826,E2 -16825.826} C_VEL
LIN {X 0,Y 289.451,Z 688.094,A -85,B 0,C 180,E1 -16828.609,E2 -16828.609} C_VEL
LIN {X 0,Y 289.43,Z 688.327,A -85,B 0,C 180,E1 -16830,E2 -16830} C_VEL
LIN {X 0,Y 289.451,Z 688.132,A -85,B 0,C 180,E1 -16831.391,E2 -16831.391} C_VEL
LIN {X 0,Y 289.686,Z 686.574,A -85,B 0,C 180,E1 -16834.174,E2 -16834.174} C_VEL
LIN {X 0,Y 289.996,Z 684.075,A -85,B 0,C 180,E1 -16836.469,E2 -16836.469} C_VEL
LIN {X 0,Y 290.384,Z 681.122,A -85,B 0,C 180,E1 -16838.35,E2 -16838.35} C_VEL
LIN {X 0,Y 291.101,Z 676.843,A -85,B 0,C 180,E1 -16840.432,E2 -16840.432} C_VEL
LIN {X 0,Y 292.089,Z 671.374,A -85,B 0,C 180,E1 -16842.507,E2 -16842.507} C_VEL
LIN {X 0,Y 293.352,Z 664.512,A -85,B 0,C 180,E1 -16844.57,E2 -16844.57} C_VEL
LIN {X 0,Y 294.995,Z 655.925,A -85,B 0,C 180,E1 -16846.612,E2 -16846.612} C_VEL
LIN {X 0,Y 296.549,Z 646.765,A -85,B 0,C 180,E1 -16848.369,E2 -16848.369} C_VEL
LIN {X 0,Y 298.071,Z 636.187,A -85,B 0,C 180,E1 -16849.992,E2 -16849.992} C_VEL
LIN {X 0,Y 299.654,Z 625.172,A -85,B 0,C 180,E1 -16851.317,E2 -16851.317} C_VEL
LIN {X 0,Y 300.843,Z 614.76,A -85,B 0,C 180,E1 -16852.31,E2 -16852.31} C_VEL
LIN {X 0,Y 302.035,Z 603.563,A -85,B 0,C 180,E1 -16853.12,E2 -16853.12} C_VEL
LIN {X 0,Y 302.815,Z 590.899,A -85,B 0,C 180,E1 -16853.782,E2 -16853.782} C_VEL
LIN {X 0,Y 303.482,Z 576.265,A -85,B 0,C 180,E1 -16854.226,E2 -16854.226} C_VEL
LIN {X 0,Y 305.159,Z 506.323,A -85,B 0,C 180,E1 -16855.871,E2 -16855.871} C_VEL
LIN {X 0,Y 300.193,Z 478.335,A -85,B 0,C 180,E1 -16857.07,E2 -16857.07} C_VEL
LIN {X 0,Y 299.352,Z 473.715,A -85,B 0,C 180,E1 -16857.313,E2 -16857.313} C_VEL
LIN {X 0,Y 299.512,Z 470.274,A -85,B 0,C 180,E1 -16857.989,E2 -16857.989} C_VEL
LIN {X 0,Y 297.35,Z 459.4,A -85,B 0,C 180,E1 -16860.533,E2 -16860.533} C_VEL
LIN {X 0,Y 296.804,Z 457.027,A -85,B 0,C 180,E1 -16861.125,E2 -16861.125} C_VEL
LIN {X 0,Y 295.373,Z 453.74,A -85,B 0,C 180,E1 -16862.031,E2 -16862.031} C_VEL
LIN {X 0,Y 291.271,Z 449.224,A -85,B 0,C 180,E1 -16863.559,E2 -16863.559} C_VEL
LIN {X 0,Y 287.782,Z 445.741,A -85,B 0,C 180,E1 -16864.811,E2 -16864.811} C_VEL
LIN {X 0,Y 285.831,Z 442.757,A -85,B 0,C 180,E1 -16865.768,E2 -16865.768} C_VEL
LIN {X 0,Y 285.413,Z 441.631,A -85,B 0,C 180,E1 -16866.087,E2 -16866.087} C_VEL
LIN {X 0,Y 284.376,Z 438.059,A -85,B 0,C 180,E1 -16867.097,E2 -16867.097} C_VEL
LIN {X 0,Y 284.31,Z 438.063,A -85,B 0,C 180,E1 -16869.994,E2 -16869.994} C_VEL
LIN {X 0,Y 284.279,Z 438.066,A -85,B 0,C 180,E1 -16874.197,E2 -16874.197} C_VEL
LIN {X 0,Y 284.274,Z 438.062,A -85,B 0,C 180,E1 -16878.124,E2 -16878.124} C_VEL
LIN {X 0,Y 284.329,Z 438.056,A -85,B 0,C 180,E1 -16882.277,E2 -16882.277} C_VEL
LIN {X 0,Y 284.312,Z 438.065,A -85,B 0,C 180,E1 -16885.351,E2 -16885.351} C_VEL
LIN {X 0,Y 284.367,Z 438.261,A -85,B 0,C 180,E1 -16887.693,E2 -16887.693} C_VEL
LIN {X 0,Y 288.176,Z 456.031,A -85,B 0,C 180,E1 -16891.856,E2 -16891.856} C_VEL
LIN {X 0,Y 289.316,Z 462.666,A -85,B 0,C 180,E1 -16893.373,E2 -16893.373} C_VEL
LIN {X 0,Y 288.582,Z 472.891,A -85,B 0,C 180,E1 -16895.543,E2 -16895.543} C_VEL
LIN {X 0,Y 288.413,Z 474.711,A -85,B 0,C 180,E1 -16895.922,E2 -16895.922} C_VEL
LIN {X 0,Y 291.527,Z 502.463,A -85,B 0,C 180,E1 -16897.117,E2 -16897.117} C_VEL
LIN {X 0,Y 291.728,Z 507.16,A -85,B 0,C 180,E1 -16897.301,E2 -16897.301} C_VEL
LIN {X 0,Y 288.84,Z 586.79,A -85,B 0,C 180,E1 -16900.223,E2 -16900.223} C_VEL
LIN {X 0,Y 288.169,Z 601.124,A -85,B 0,C 180,E1 -16901.054,E2 -16901.054} C_VEL
LIN {X 0,Y 287.223,Z 615.025,A -85,B 0,C 180,E1 -16902.19,E2 -16902.19} C_VEL
LIN {X 0,Y 286.266,Z 627.466,A -85,B 0,C 180,E1 -16903.521,E2 -16903.521} C_VEL
LIN {X 0,Y 285.538,Z 637.375,A -85,B 0,C 180,E1 -16904.84,E2 -16904.84} C_VEL
LIN {X 0,Y 284.74,Z 647.326,A -85,B 0,C 180,E1 -16906.439,E2 -16906.439} C_VEL
LIN {X 0,Y 283.836,Z 657.997,A -85,B 0,C 180,E1 -16908.575,E2 -16908.575} C_VEL
LIN {X 0,Y 283.219,Z 666.533,A -85,B 0,C 180,E1 -16910.718,E2 -16910.718} C_VEL
LIN {X 0,Y 282.744,Z 673.388,A -85,B 0,C 180,E1 -16912.861,E2 -16912.861} C_VEL
LIN {X 0,Y 282.499,Z 678.44,A -85,B 0,C 180,E1 -16914.835,E2 -16914.835} C_VEL
LIN {X 0,Y 282.456,Z 682.991,A -85,B 0,C 180,E1 -16917.148,E2 -16917.148} C_VEL
LIN {X 0,Y 282.348,Z 685.102,A -85,B 0,C 180,E1 -16918.574,E2 -16918.574} C_VEL
LIN {X 0,Y 282.343,Z 686.783,A -85,B 0,C 180,E1 -16920,E2 -16920} C_VEL
LIN {X 0,Y 282.396,Z 687.979,A -85,B 0,C 180,E1 -16921.426,E2 -16921.426} C_VEL
LIN {X 0,Y 282.52,Z 688.746,A -85,B 0,C 180,E1 -16922.852,E2 -16922.852} C_VEL
LIN {X 0,Y 282.694,Z 689.106,A -85,B 0,C 180,E1 -16924.277,E2 -16924.277} C_VEL
LIN {X 0,Y 283.004,Z 688.995,A -85,B 0,C 180,E1 -16925.701,E2 -16925.701} C_VEL
LIN {X 0,Y 283.408,Z 688.381,A -85,B 0,C 180,E1 -16927.283,E2 -16927.283} C_VEL
LIN {X 0,Y 284.454,Z 686.154,A -85,B 0,C 180,E1 -16929.959,E2 -16929.959} C_VEL
LIN {X 0,Y 285.672,Z 683.244,A -85,B 0,C 180,E1 -16932.07,E2 -16932.07} C_VEL
LIN {X 0,Y 287.108,Z 679.277,A -85,B 0,C 180,E1 -16934.169,E2 -16934.169} C_VEL
LIN {X 0,Y 289.179,Z 674.151,A -85,B 0,C 180,E1 -16936.23,E2 -16936.23} C_VEL
LIN {X 0,Y 291.422,Z 667.751,A -85,B 0,C 180,E1 -16938.271,E2 -16938.271} C_VEL
LIN {X 0,Y 294.103,Z 659.806,A -85,B 0,C 180,E1 -16940.273,E2 -16940.273} C_VEL
LIN {X 0,Y 297.141,Z 650.075,A -85,B 0,C 180,E1 -16942.237,E2 -16942.237} C_VEL
LIN {X 0,Y 299.991,Z 639.865,A -85,B 0,C 180,E1 -16943.873,E2 -16943.873} C_VEL
LIN {X 0,Y 303.016,Z 627.886,A -85,B 0,C 180,E1 -16945.409,E2 -16945.409} C_VEL
LIN {X 0,Y 305.666,Z 615.679,A -85,B 0,C 180,E1 -16946.638,E2 -16946.638} C_VEL
LIN {X 0,Y 307.977,Z 603.027,A -85,B 0,C 180,E1 -16947.615,E2 -16947.615} C_VEL
LIN {X 0,Y 310.026,Z 589.458,A -85,B 0,C 180,E1 -16948.382,E2 -16948.382} C_VEL
LIN {X 0,Y 318.992,Z 516.963,A -85,B 0,C 180,E1 -16951.391,E2 -16951.391} C_VEL
LIN {X 0,Y 317.804,Z 504.486,A -85,B 0,C 180,E1 -16952.761,E2 -16952.761} C_VEL
LIN {X 0,Y 317.439,Z 502.609,A -85,B 0,C 180,E1 -16953.044,E2 -16953.044} C_VEL
LIN {X 0,Y 315.474,Z 497.701,A -85,B 0,C 180,E1 -16954.171,E2 -16954.171} C_VEL
LIN {X 0,Y 313.627,Z 493.482,A -85,B 0,C 180,E1 -16955.333,E2 -16955.333} C_VEL
LIN {X 0,Y 311.758,Z 489.481,A -85,B 0,C 180,E1 -16956.672,E2 -16956.672} C_VEL
LIN {X 0,Y 309.593,Z 485.021,A -85,B 0,C 180,E1 -16958.58,E2 -16958.58} C_VEL
LIN {X 0,Y 307.534,Z 481.217,A -85,B 0,C 180,E1 -16961.13,E2 -16961.13} C_VEL
LIN {X 0,Y 307.085,Z 480.077,A -85,B 0,C 180,E1 -16962.175,E2 -16962.175} C_VEL
LIN {X 0,Y 307.23,Z 478.916,A -85,B 0,C 180,E1 -16964.835,E2 -16964.835} C_VEL
LIN {X 0,Y 307.82,Z 478.927,A -85,B 0,C 180,E1 -16966.938,E2 -16966.938} C_VEL
LIN {X 0,Y 308.614,Z 479.623,A -85,B 0,C 180,E1 -16968.721,E2 -16968.721} C_VEL
LIN {X 0,Y 310.615,Z 481.866,A -85,B 0,C 180,E1 -16971.426,E2 -16971.426} C_VEL
LIN {X 0,Y 312.548,Z 484.297,A -85,B 0,C 180,E1 -16972.916,E2 -16972.916} C_VEL
LIN {X 0,Y 314.141,Z 486.835,A -85,B 0,C 180,E1 -16974.009,E2 -16974.009} C_VEL
LIN {X 0,Y 315.826,Z 494.132,A -85,B 0,C 180,E1 -16975.508,E2 -16975.508} C_VEL
LIN {X 0,Y 316.439,Z 508.17,A -85,B 0,C 180,E1 -16977.047,E2 -16977.047} C_VEL
LIN {X 0,Y 316.652,Z 523.547,A -85,B 0,C 180,E1 -16978.399,E2 -16978.399} C_VEL
LIN {X 0,Y 316.152,Z 535.541,A -85,B 0,C 180,E1 -16979.213,E2 -16979.213} C_VEL
LIN {X 0,Y 315.406,Z 542.864,A -85,B 0,C 180,E1 -16979.569,E2 -16979.569} C_VEL
LIN {X 0,Y 307.508,Z 605.973,A -85,B 0,C 180,E1 -16982.247,E2 -16982.247} C_VEL
LIN {X 0,Y 305.264,Z 619.165,A -85,B 0,C 180,E1 -16983.047,E2 -16983.047} C_VEL
LIN {X 0,Y 302.426,Z 632.889,A -85,B 0,C 180,E1 -16984.168,E2 -16984.168} C_VEL
LIN {X 0,Y 299.347,Z 645.714,A -85,B 0,C 180,E1 -16985.556,E2 -16985.556} C_VEL
LIN {X 0,Y 296.549,Z 656.058,A -85,B 0,C 180,E1 -16986.981,E2 -16986.981} C_VEL
LIN {X 0,Y 293.374,Z 667.348,A -85,B 0,C 180,E1 -16988.94,E2 -16988.94} C_VEL
LIN {X 0,Y 290.73,Z 676.005,A -85,B 0,C 180,E1 -16990.848,E2 -16990.848} C_VEL
LIN {X 0,Y 288.181,Z 683.823,A -85,B 0,C 180,E1 -16992.983,E2 -16992.983} C_VEL
LIN {X 0,Y 286.356,Z 689.806,A -85,B 0,C 180,E1 -16995.066,E2 -16995.066} C_VEL
LIN {X 0,Y 284.884,Z 694.526,A -85,B 0,C 180,E1 -16997.172,E2 -16997.172} C_VEL
LIN {X 0,Y 283.768,Z 698.167,A -85,B 0,C 180,E1 -16999.295,E2 -16999.295} C_VEL
LIN {X 0,Y 283.01,Z 700.763,A -85,B 0,C 180,E1 -17001.431,E2 -17001.431} C_VEL
LIN {X 0,Y 282.666,Z 701.92,A -85,B 0,C 180,E1 -17002.859,E2 -17002.859} C_VEL
LIN {X 0,Y 282.461,Z 702.723,A -85,B 0,C 180,E1 -17004.416,E2 -17004.416} C_VEL
LIN {X 0,Y 282.407,Z 702.988,A -85,B 0,C 180,E1 -17005.718,E2 -17005.718} C_VEL
LIN {X 0,Y 282.433,Z 702.833,A -85,B 0,C 180,E1 -17007.147,E2 -17007.147} C_VEL
LIN {X 0,Y 282.41,Z 703.559,A -85,B 0,C 180,E1 -17010,E2 -17010} C_VEL
LIN {X 0,Y 282.381,Z 703.333,A -85,B 0,C 180,E1 -17011.426,E2 -17011.426} C_VEL
LIN {X 0,Y 282.409,Z 702.713,A -85,B 0,C 180,E1 -17012.853,E2 -17012.853} C_VEL
LIN {X 0,Y 282.415,Z 700.518,A -85,B 0,C 180,E1 -17015.487,E2 -17015.487} C_VEL
LIN {X 0,Y 282.698,Z 697.277,A -85,B 0,C 180,E1 -17017.859,E2 -17017.859} C_VEL
LIN {X 0,Y 283.194,Z 693.228,A -85,B 0,C 180,E1 -17020.004,E2 -17020.004} C_VEL
LIN {X 0,Y 284.092,Z 686.988,A -85,B 0,C 180,E1 -17022.501,E2 -17022.501} C_VEL
LIN {X 0,Y 285.366,Z 680.188,A -85,B 0,C 180,E1 -17024.622,E2 -17024.622} C_VEL
LIN {X 0,Y 286.58,Z 673.226,A -85,B 0,C 180,E1 -17026.381,E2 -17026.381} C_VEL
LIN {X 0,Y 288.034,Z 664.499,A -85,B 0,C 180,E1 -17028.187,E2 -17028.187} C_VEL
LIN {X 0,Y 288.969,Z 658.907,A -85,B 0,C 180,E1 -17029.168,E2 -17029.168} C_VEL
LIN {X 0,Y 291.757,Z 649.846,A -85,B 0,C 180,E1 -17031.182,E2 -17031.182} C_VEL
LIN {X 0,Y 294.809,Z 639.798,A -85,B 0,C 180,E1 -17032.977,E2 -17032.977} C_VEL
LIN {X 0,Y 297.941,Z 628.854,A -85,B 0,C 180,E1 -17034.567,E2 -17034.567} C_VEL
LIN {X 0,Y 301.227,Z 616.812,A -85,B 0,C 180,E1 -17035.942,E2 -17035.942} C_VEL
LIN {X 0,Y 304.384,Z 603.683,A -85,B 0,C 180,E1 -17037.13,E2 -17037.13} C_VEL
LIN {X 0,Y 307.638,Z 587.673,A -85,B 0,C 180,E1 -17038.204,E2 -17038.204} C_VEL
LIN {X 0,Y 309.81,Z 573.095,A -85,B 0,C 180,E1 -17038.913,E2 -17038.913} C_VEL
LIN {X 0,Y 314.124,Z 534.922,A -85,B 0,C 180,E1 -17040.505,E2 -17040.505} C_VEL
LIN {X 0,Y 314.275,Z 523.266,A -85,B 0,C 180,E1 -17041.302,E2 -17041.302} C_VEL
LIN {X 0,Y 313.862,Z 511.943,A -85,B 0,C 180,E1 -17042.278,E2 -17042.278} C_VEL
LIN {X 0,Y 312.93,Z 499.072,A -85,B 0,C 180,E1 -17043.62,E2 -17043.62} C_VEL
LIN {X 0,Y 312.407,Z 494.83,A -85,B 0,C 180,E1 -17044.169,E2 -17044.169} C_VEL
LIN {X 0,Y 310.977,Z 490.887,A -85,B 0,C 180,E1 -17045.045,E2 -17045.045} C_VEL
LIN {X 0,Y 308.835,Z 485.257,A -85,B 0,C 180,E1 -17046.487,E2 -17046.487} C_VEL
LIN {X 0,Y 305.878,Z 478.069,A -85,B 0,C 180,E1 -17048.916,E2 -17048.916} C_VEL
LIN {X 0,Y 303.51,Z 473.063,A -85,B 0,C 180,E1 -17051.635,E2 -17051.635} C_VEL
LIN {X 0,Y 302.507,Z 470.159,A -85,B 0,C 180,E1 -17053.928,E2 -17053.928} C_VEL
LIN {X 0,Y 302.368,Z 468.629,A -85,B 0,C 180,E1 -17056.099,E2 -17056.099} C_VEL
LIN {X 0,Y 302.865,Z 468.169,A -85,B 0,C 180,E1 -17057.95,E2 -17057.95} C_VEL
LIN {X 0,Y 304.428,Z 468.334,A -85,B 0,C 180,E1 -17060.307,E2 -17060.307} C_VEL
LIN {X 0,Y 307.425,Z 471.131,A -85,B 0,C 180,E1 -17063.143,E2 -17063.143} C_VEL
LIN {X 0,Y 310.537,Z 474.697,A -85,B 0,C 180,E1 -17065.227,E2 -17065.227} C_VEL
LIN {X 0,Y 312.968,Z 477.957,A -85,B 0,C 180,E1 -17066.595,E2 -17066.595} C_VEL
LIN {X 0,Y 315.902,Z 482.093,A -85,B 0,C 180,E1 -17068.013,E2 -17068.013} C_VEL
LIN {X 0,Y 318.814,Z 486.94,A -85,B 0,C 180,E1 -17069.286,E2 -17069.286} C_VEL
LIN {X 0,Y 312.457,Z 537.717,A -85,B 0,C 180,E1 -17071.447,E2 -17071.447} C_VEL
LIN {X 0,Y 310.887,Z 550.934,A -85,B 0,C 180,E1 -17072.165,E2 -17072.165} C_VEL
LIN {X 0,Y 309.01,Z 563.706,A -85,B 0,C 180,E1 -17073.125,E2 -17073.125} C_VEL
LIN {X 0,Y 306.551,Z 576.512,A -85,B 0,C 180,E1 -17074.359,E2 -17074.359} C_VEL
LIN {X 0,Y 303.877,Z 587.925,A -85,B 0,C 180,E1 -17075.763,E2 -17075.763} C_VEL
LIN {X 0,Y 301.106,Z 598.225,A -85,B 0,C 180,E1 -17077.349,E2 -17077.349} C_VEL
LIN {X 0,Y 298.557,Z 606.758,A -85,B 0,C 180,E1 -17078.962,E2 -17078.962} C_VEL
LIN {X 0,Y 295.749,Z 615.051,A -85,B 0,C 180,E1 -17080.929,E2 -17080.929} C_VEL
LIN {X 0,Y 293.228,Z 621.818,A -85,B 0,C 180,E1 -17082.926,E2 -17082.926} C_VEL
LIN {X 0,Y 290.644,Z 628.005,A -85,B 0,C 180,E1 -17085.292,E2 -17085.292} C_VEL
LIN {X 0,Y 288.773,Z 631.984,A -85,B 0,C 180,E1 -17087.348,E2 -17087.348} C_VEL
LIN {X 0,Y 287.617,Z 634.069,A -85,B 0,C 180,E1 -17088.727,E2 -17088.727} C_VEL
LIN {X 0,Y 286.602,Z 635.721,A -85,B 0,C 180,E1 -17090.116,E2 -17090.116} C_VEL
LIN {X 0,Y 285.786,Z 636.894,A -85,B 0,C 180,E1 -17091.515,E2 -17091.515} C_VEL
LIN {X 0,Y 285.127,Z 637.617,A -85,B 0,C 180,E1 -17092.921,E2 -17092.921} C_VEL
LIN {X 0,Y 284.542,Z 637.942,A -85,B 0,C 180,E1 -17094.33,E2 -17094.33} C_VEL
LIN {X 0,Y 284.03,Z 637.864,A -85,B 0,C 180,E1 -17095.743,E2 -17095.743} C_VEL
LIN {X 0,Y 283.616,Z 637.328,A -85,B 0,C 180,E1 -17097.159,E2 -17097.159} C_VEL
LIN {X 0,Y 283.319,Z 636.366,A -85,B 0,C 180,E1 -17098.579,E2 -17098.579} C_VEL
LIN {X 0,Y 283.166,Z 634.99,A -85,B 0,C 180,E1 -17100,E2 -17100} C_VEL
LIN {X 0,Y 283.167,Z 632.072,A -85,B 0,C 180,E1 -17102.134,E2 -17102.134} C_VEL
LIN {X 0,Y 283.3,Z 628.107,A -85,B 0,C 180,E1 -17104.268,E2 -17104.268} C_VEL
LIN {X 0,Y 283.523,Z 622.982,A -85,B 0,C 180,E1 -17106.405,E2 -17106.405} C_VEL
LIN {X 0,Y 283.904,Z 615.238,A -85,B 0,C 180,E1 -17108.901,E2 -17108.901} C_VEL
LIN {X 0,Y 284.504,Z 606.907,A -85,B 0,C 180,E1 -17111.037,E2 -17111.037} C_VEL
LIN {X 0,Y 285.191,Z 598.408,A -85,B 0,C 180,E1 -17112.814,E2 -17112.814} C_VEL
LIN {X 0,Y 286.032,Z 588.13,A -85,B 0,C 180,E1 -17114.587,E2 -17114.587} C_VEL
LIN {X 0,Y 286.814,Z 576.738,A -85,B 0,C 180,E1 -17116.185,E2 -17116.185} C_VEL
LIN {X 0,Y 287.642,Z 565.047,A -85,B 0,C 180,E1 -17117.499,E2 -17117.499} C_VEL
LIN {X 0,Y 288.348,Z 551.962,A -85,B 0,C 180,E1 -17118.657,E2 -17118.657} C_VEL
LIN {X 0,Y 289.075,Z 537.008,A -85,B 0,C 180,E1 -17119.622,E2 -17119.622} C_VEL
LIN {X 0,Y 289.511,Z 520.177,A -85,B 0,C 180,E1 -17120.331,E2 -17120.331} C_VEL
LIN {X 0,Y 291.527,Z 461.205,A -85,B 0,C 180,E1 -17122.481,E2 -17122.481} C_VEL
LIN {X 0,Y 284.35,Z 438.057,A -85,B 0,C 180,E1 -17123.706,E2 -17123.706} C_VEL
LIN {X 0,Y 284.394,Z 438.053,A -85,B 0,C 180,E1 -17127.172,E2 -17127.172} C_VEL
LIN {X 0,Y 284.296,Z 438.064,A -85,B 0,C 180,E1 -17131.274,E2 -17131.274} C_VEL
LIN {X 0,Y 284.343,Z 438.049,A -85,B 0,C 180,E1 -17135.348,E2 -17135.348} C_VEL
LIN {X 0,Y 284.321,Z 438.071,A -85,B 0,C 180,E1 -17138.168,E2 -17138.168} C_VEL
LIN {X 0,Y 284.271,Z 438.07,A -85,B 0,C 180,E1 -17142.124,E2 -17142.124} C_VEL
LIN {X 0,Y 284.256,Z 438.061,A -85,B 0,C 180,E1 -17146.189,E2 -17146.189} C_VEL
LIN {X 0,Y 284.309,Z 438.059,A -85,B 0,C 180,E1 -17150.024,E2 -17150.024} C_VEL
LIN {X 0,Y 284.393,Z 438.169,A -85,B 0,C 180,E1 -17153.099,E2 -17153.099} C_VEL
LIN {X 0,Y 287.919,Z 450.464,A -85,B 0,C 180,E1 -17156.471,E2 -17156.471} C_VEL
LIN {X 0,Y 290.862,Z 462.379,A -85,B 0,C 180,E1 -17159.508,E2 -17159.508} C_VEL
LIN {X 0,Y 292.836,Z 472.158,A -85,B 0,C 180,E1 -17161.807,E2 -17161.807} C_VEL
LIN {X 0,Y 292.858,Z 474.427,A -85,B 0,C 180,E1 -17162.207,E2 -17162.207} C_VEL
LIN {X 0,Y 297.655,Z 500.64,A -85,B 0,C 180,E1 -17163.393,E2 -17163.393} C_VEL
LIN {X 0,Y 298.767,Z 507.931,A -85,B 0,C 180,E1 -17163.692,E2 -17163.692} C_VEL
LIN {X 0,Y 296.921,Z 578.925,A -85,B 0,C 180,E1 -17165.39,E2 -17165.39} C_VEL
LIN {X 0,Y 296.275,Z 592.512,A -85,B 0,C 180,E1 -17165.846,E2 -17165.846} C_VEL
LIN {X 0,Y 295.307,Z 604.611,A -85,B 0,C 180,E1 -17166.507,E2 -17166.507} C_VEL
LIN {X 0,Y 294.039,Z 617.509,A -85,B 0,C 180,E1 -17167.516,E2 -17167.516} C_VEL
LIN {X 0,Y 292.523,Z 628.908,A -85,B 0,C 180,E1 -17168.692,E2 -17168.692} C_VEL
LIN {X 0,Y 290.796,Z 640.313,A -85,B 0,C 180,E1 -17170.223,E2 -17170.223} C_VEL
LIN {X 0,Y 289.205,Z 650.478,A -85,B 0,C 180,E1 -17171.95,E2 -17171.95} C_VEL
LIN {X 0,Y 287.334,Z 660.173,A -85,B 0,C 180,E1 -17174.028,E2 -17174.028} C_VEL
LIN {X 0,Y 285.824,Z 667.96,A -85,B 0,C 180,E1 -17176.129,E2 -17176.129} C_VEL
LIN {X 0,Y 284.817,Z 673.218,A -85,B 0,C 180,E1 -17177.893,E2 -17177.893} C_VEL
LIN {X 0,Y 283.84,Z 678.354,A -85,B 0,C 180,E1 -17180.019,E2 -17180.019} C_VEL
LIN {X 0,Y 283.211,Z 682.327,A -85,B 0,C 180,E1 -17182.155,E2 -17182.155} C_VEL
LIN {X 0,Y 282.765,Z 685.256,A -85,B 0,C 180,E1 -17184.294,E2 -17184.294} C_VEL
LIN {X 0,Y 282.61,Z 686.674,A -85,B 0,C 180,E1 -17185.721,E2 -17185.721} C_VEL
LIN {X 0,Y 282.479,Z 687.669,A -85,B 0,C 180,E1 -17187.148,E2 -17187.148} C_VEL
LIN {X 0,Y 282.351,Z 688.516,A -85,B 0,C 180,E1 -17190,E2 -17190} C_VEL
LIN {X 0,Y 282.375,Z 688.321,A -85,B 0,C 180,E1 -17191.426,E2 -17191.426} C_VEL
LIN {X 0,Y 282.479,Z 687.732,A -85,B 0,C 180,E1 -17192.852,E2 -17192.852} C_VEL
LIN {X 0,Y 282.609,Z 686.762,A -85,B 0,C 180,E1 -17194.279,E2 -17194.279} C_VEL
LIN {X 0,Y 282.894,Z 684.523,A -85,B 0,C 180,E1 -17196.418,E2 -17196.418} C_VEL
LIN {X 0,Y 283.365,Z 681.309,A -85,B 0,C 180,E1 -17198.558,E2 -17198.558} C_VEL
LIN {X 0,Y 284.102,Z 677.03,A -85,B 0,C 180,E1 -17200.692,E2 -17200.692} C_VEL
LIN {X 0,Y 285.165,Z 671.559,A -85,B 0,C 180,E1 -17202.815,E2 -17202.815} C_VEL
LIN {X 0,Y 286.48,Z 664.695,A -85,B 0,C 180,E1 -17204.927,E2 -17204.927} C_VEL
LIN {X 0,Y 288.207,Z 656.105,A -85,B 0,C 180,E1 -17207.015,E2 -17207.015} C_VEL
LIN {X 0,Y 289.717,Z 647.515,A -85,B 0,C 180,E1 -17208.708,E2 -17208.708} C_VEL
LIN {X 0,Y 291.236,Z 637.607,A -85,B 0,C 180,E1 -17210.297,E2 -17210.297} C_VEL
LIN {X 0,Y 292.874,Z 626.863,A -85,B 0,C 180,E1 -17211.651,E2 -17211.651} C_VEL
LIN {X 0,Y 294.31,Z 614.92,A -85,B 0,C 180,E1 -17212.833,E2 -17212.833} C_VEL
LIN {X 0,Y 295.598,Z 602.342,A -85,B 0,C 180,E1 -17213.747,E2 -17213.747} C_VEL
LIN {X 0,Y 296.447,Z 588.957,A -85,B 0,C 180,E1 -17214.419,E2 -17214.419} C_VEL
LIN {X 0,Y 297.144,Z 572.758,A -85,B 0,C 180,E1 -17214.87,E2 -17214.87} C_VEL
LIN {X 0,Y 298.793,Z 507.422,A -85,B 0,C 180,E1 -17216.437,E2 -17216.437} C_VEL
LIN {X 0,Y 293.864,Z 479.593,A -85,B 0,C 180,E1 -17217.67,E2 -17217.67} C_VEL
LIN {X 0,Y 292.831,Z 473.806,A -85,B 0,C 180,E1 -17217.983,E2 -17217.983} C_VEL
LIN {X 0,Y 292.522,Z 470.36,A -85,B 0,C 180,E1 -17218.719,E2 -17218.719} C_VEL
LIN {X 0,Y 290.156,Z 458.997,A -85,B 0,C 180,E1 -17221.464,E2 -17221.464} C_VEL
LIN {X 0,Y 286.85,Z 446.573,A -85,B 0,C 180,E1 -17224.711,E2 -17224.711} C_VEL
LIN {X 0,Y 285.413,Z 441.631,A -85,B 0,C 180,E1 -17226.087,E2 -17226.087} C_VEL
LIN {X 0,Y 284.509,Z 439.88,A -85,B 0,C 180,E1 -17226.747,E2 -17226.747} C_VEL
LIN {X 0,Y 283.296,Z 438.938,A -85,B 0,C 180,E1 -17227.462,E2 -17227.462} C_VEL
LIN {X 0,Y 280.582,Z 438.536,A -85,B 0,C 180,E1 -17228.967,E2 -17228.967} C_VEL
LIN {X 0,Y 278.206,Z 438.823,A -85,B 0,C 180,E1 -17230.578,E2 -17230.578} C_VEL
LIN {X 0,Y 277.278,Z 438.949,A -85,B 0,C 180,E1 -17231.828,E2 -17231.828} C_VEL
LIN {X 0,Y 277.218,Z 438.948,A -85,B 0,C 180,E1 -17232.25,E2 -17232.25} C_VEL
LIN {X 0,Y 277.222,Z 438.953,A -85,B 0,C 180,E1 -17235.222,E2 -17235.222} C_VEL
LIN {X 0,Y 277.224,Z 438.948,A -85,B 0,C 180,E1 -17239.512,E2 -17239.512} C_VEL
LIN {X 0,Y 277.274,Z 438.932,A -85,B 0,C 180,E1 -17242.531,E2 -17242.531} C_VEL
LIN {X 0,Y 277.253,Z 438.948,A -85,B 0,C 180,E1 -17246.105,E2 -17246.105} C_VEL
LIN {X 0,Y 277.329,Z 439.108,A -85,B 0,C 180,E1 -17247.393,E2 -17247.393} C_VEL
LIN {X 0,Y 281.141,Z 456.923,A -85,B 0,C 180,E1 -17251.643,E2 -17251.643} C_VEL
LIN {X 0,Y 282.215,Z 462.616,A -85,B 0,C 180,E1 -17252.968,E2 -17252.968} C_VEL
LIN {X 0,Y 281.967,Z 470.014,A -85,B 0,C 180,E1 -17254.578,E2 -17254.578} C_VEL
LIN {X 0,Y 281.477,Z 474.823,A -85,B 0,C 180,E1 -17255.608,E2 -17255.608} C_VEL
LIN {X 0,Y 284.351,Z 501.546,A -85,B 0,C 180,E1 -17256.783,E2 -17256.783} C_VEL
LIN {X 0,Y 284.817,Z 506.15,A -85,B 0,C 180,E1 -17256.981,E2 -17256.981} C_VEL
LIN {X 0,Y 281.83,Z 586.181,A -85,B 0,C 180,E1 -17260.042,E2 -17260.042} C_VEL
LIN {X 0,Y 281.161,Z 599.998,A -85,B 0,C 180,E1 -17260.848,E2 -17260.848} C_VEL
LIN {X 0,Y 280.262,Z 613.297,A -85,B 0,C 180,E1 -17261.921,E2 -17261.921} C_VEL
LIN {X 0,Y 279.367,Z 625.643,A -85,B 0,C 180,E1 -17263.221,E2 -17263.221} C_VEL
LIN {X 0,Y 278.559,Z 636.353,A -85,B 0,C 180,E1 -17264.638,E2 -17264.638} C_VEL
LIN {X 0,Y 277.612,Z 647.527,A -85,B 0,C 180,E1 -17266.457,E2 -17266.457} C_VEL
LIN {X 0,Y 276.722,Z 658.221,A -85,B 0,C 180,E1 -17268.648,E2 -17268.648} C_VEL
LIN {X 0,Y 276.09,Z 666.768,A -85,B 0,C 180,E1 -17270.845,E2 -17270.845} C_VEL
LIN {X 0,Y 275.631,Z 673.603,A -85,B 0,C 180,E1 -17273.043,E2 -17273.043} C_VEL
LIN {X 0,Y 275.403,Z 678.325,A -85,B 0,C 180,E1 -17274.936,E2 -17274.936} C_VEL
LIN {X 0,Y 275.388,Z 682.562,A -85,B 0,C 180,E1 -17277.074,E2 -17277.074} C_VEL
LIN {X 0,Y 275.275,Z 684.82,A -85,B 0,C 180,E1 -17278.537,E2 -17278.537} C_VEL
LIN {X 0,Y 275.266,Z 686.596,A -85,B 0,C 180,E1 -17280,E2 -17280} C_VEL
LIN {X 0,Y 275.321,Z 687.952,A -85,B 0,C 180,E1 -17281.463,E2 -17281.463} C_VEL
LIN {X 0,Y 275.433,Z 688.829,A -85,B 0,C 180,E1 -17282.925,E2 -17282.925} C_VEL
LIN {X 0,Y 275.626,Z 689.277,A -85,B 0,C 180,E1 -17284.387,E2 -17284.387} C_VEL
LIN {X 0,Y 275.938,Z 689.321,A -85,B 0,C 180,E1 -17285.847,E2 -17285.847} C_VEL
LIN {X 0,Y 276.337,Z 688.918,A -85,B 0,C 180,E1 -17287.306,E2 -17287.306} C_VEL
LIN {X 0,Y 276.82,Z 688.085,A -85,B 0,C 180,E1 -17288.762,E2 -17288.762} C_VEL
LIN {X 0,Y 277.501,Z 686.84,A -85,B 0,C 180,E1 -17290.211,E2 -17290.211} C_VEL
LIN {X 0,Y 278.799,Z 684.147,A -85,B 0,C 180,E1 -17292.373,E2 -17292.373} C_VEL
LIN {X 0,Y 280.325,Z 680.45,A -85,B 0,C 180,E1 -17294.519,E2 -17294.519} C_VEL
LIN {X 0,Y 282.528,Z 675.555,A -85,B 0,C 180,E1 -17296.623,E2 -17296.623} C_VEL
LIN {X 0,Y 285.283,Z 668.318,A -85,B 0,C 180,E1 -17299.051,E2 -17299.051} C_VEL
LIN {X 0,Y 288.203,Z 660.517,A -85,B 0,C 180,E1 -17301.081,E2 -17301.081} C_VEL
LIN {X 0,Y 291.534,Z 650.554,A -85,B 0,C 180,E1 -17303.127,E2 -17303.127} C_VEL
LIN {X 0,Y 294.587,Z 640.652,A -85,B 0,C 180,E1 -17304.761,E2 -17304.761} C_VEL
LIN {X 0,Y 297.574,Z 629.724,A -85,B 0,C 180,E1 -17306.205,E2 -17306.205} C_VEL
LIN {X 0,Y 300.515,Z 617.278,A -85,B 0,C 180,E1 -17307.509,E2 -17307.509} C_VEL
LIN {X 0,Y 302.987,Z 605.315,A -85,B 0,C 180,E1 -17308.487,E2 -17308.487} C_VEL
LIN {X 0,Y 305.121,Z 592.621,A -85,B 0,C 180,E1 -17309.258,E2 -17309.258} C_VEL
LIN {X 0,Y 314.923,Z 518.862,A -85,B 0,C 180,E1 -17312.418,E2 -17312.418} C_VEL
LIN {X 0,Y 314.113,Z 507.791,A -85,B 0,C 180,E1 -17313.691,E2 -17313.691} C_VEL
LIN {X 0,Y 312.342,Z 502.936,A -85,B 0,C 180,E1 -17314.849,E2 -17314.849} C_VEL
LIN {X 0,Y 310.205,Z 497.642,A -85,B 0,C 180,E1 -17316.397,E2 -17316.397} C_VEL
LIN {X 0,Y 307.575,Z 491.811,A -85,B 0,C 180,E1 -17318.75,E2 -17318.75} C_VEL
LIN {X 0,Y 305.582,Z 487.82,A -85,B 0,C 180,E1 -17321.461,E2 -17321.461} C_VEL
LIN {X 0,Y 304.96,Z 486.289,A -85,B 0,C 180,E1 -17323.193,E2 -17323.193} C_VEL
LIN {X 0,Y 304.863,Z 485.471,A -85,B 0,C 180,E1 -17325.614,E2 -17325.614} C_VEL
LIN {X 0,Y 305.703,Z 485.929,A -85,B 0,C 180,E1 -17327.902,E2 -17327.902} C_VEL
LIN {X 0,Y 307.667,Z 487.691,A -85,B 0,C 180,E1 -17330.402,E2 -17330.402} C_VEL
LIN {X 0,Y 309.574,Z 489.779,A -85,B 0,C 180,E1 -17332.067,E2 -17332.067} C_VEL
LIN {X 0,Y 311.419,Z 492.778,A -85,B 0,C 180,E1 -17333.474,E2 -17333.474} C_VEL
LIN {X 0,Y 312.565,Z 498.521,A -85,B 0,C 180,E1 -17334.67,E2 -17334.67} C_VEL
LIN {X 0,Y 312.801,Z 511.333,A -85,B 0,C 180,E1 -17336.091,E2 -17336.091} C_VEL
LIN {X 0,Y 312.68,Z 525.594,A -85,B 0,C 180,E1 -17337.395,E2 -17337.395} C_VEL
LIN {X 0,Y 311.984,Z 538.333,A -85,B 0,C 180,E1 -17338.272,E2 -17338.272} C_VEL
LIN {X 0,Y 303.034,Z 605.052,A -85,B 0,C 180,E1 -17341.186,E2 -17341.186} C_VEL
LIN {X 0,Y 300.322,Z 619.823,A -85,B 0,C 180,E1 -17342.093,E2 -17342.093} C_VEL
LIN {X 0,Y 297.511,Z 632.456,A -85,B 0,C 180,E1 -17343.142,E2 -17343.142} C_VEL
LIN {X 0,Y 294.222,Z 645.12,A -85,B 0,C 180,E1 -17344.535,E2 -17344.535} C_VEL
LIN {X 0,Y 290.909,Z 656.543,A -85,B 0,C 180,E1 -17346.13,E2 -17346.13} C_VEL
LIN {X 0,Y 288.028,Z 665.894,A -85,B 0,C 180,E1 -17347.777,E2 -17347.777} C_VEL
LIN {X 0,Y 285.006,Z 675.141,A -85,B 0,C 180,E1 -17349.804,E2 -17349.804} C_VEL
LIN {X 0,Y 282.307,Z 682.706,A -85,B 0,C 180,E1 -17351.869,E2 -17351.869} C_VEL
LIN {X 0,Y 280.088,Z 688.815,A -85,B 0,C 180,E1 -17353.978,E2 -17353.978} C_VEL
LIN {X 0,Y 278.495,Z 693.71,A -85,B 0,C 180,E1 -17356.129,E2 -17356.129} C_VEL
LIN {X 0,Y 277.129,Z 697.476,A -85,B 0,C 180,E1 -17358.295,E2 -17358.295} C_VEL
LIN {X 0,Y 276.462,Z 699.389,A -85,B 0,C 180,E1 -17359.75,E2 -17359.75} C_VEL
LIN {X 0,Y 275.976,Z 700.869,A -85,B 0,C 180,E1 -17361.211,E2 -17361.211} C_VEL
LIN {X 0,Y 275.611,Z 701.938,A -85,B 0,C 180,E1 -17362.675,E2 -17362.675} C_VEL
LIN {X 0,Y 275.367,Z 702.626,A -85,B 0,C 180,E1 -17364.485,E2 -17364.485} C_VEL
LIN {X 0,Y 275.36,Z 702.541,A -85,B 0,C 180,E1 -17367.074,E2 -17367.074} C_VEL
LIN {X 0,Y 275.311,Z 703.153,A -85,B 0,C 180,E1 -17368.537,E2 -17368.537} C_VEL
LIN {X 0,Y 275.329,Z 703.37,A -85,B 0,C 180,E1 -17370,E2 -17370} C_VEL
LIN {X 0,Y 275.304,Z 703.144,A -85,B 0,C 180,E1 -17371.463,E2 -17371.463} C_VEL
LIN {X 0,Y 275.315,Z 702.524,A -85,B 0,C 180,E1 -17372.926,E2 -17372.926} C_VEL
LIN {X 0,Y 275.335,Z 700.511,A -85,B 0,C 180,E1 -17375.445,E2 -17375.445} C_VEL
LIN {X 0,Y 275.651,Z 697.087,A -85,B 0,C 180,E1 -17378.061,E2 -17378.061} C_VEL
LIN {X 0,Y 276.179,Z 693.038,A -85,B 0,C 180,E1 -17380.261,E2 -17380.261} C_VEL
LIN {X 0,Y 277.137,Z 686.799,A -85,B 0,C 180,E1 -17382.82,E2 -17382.82} C_VEL
LIN {X 0,Y 278.485,Z 680,A -85,B 0,C 180,E1 -17384.991,E2 -17384.991} C_VEL
LIN {X 0,Y 279.768,Z 673.04,A -85,B 0,C 180,E1 -17386.792,E2 -17386.792} C_VEL
LIN {X 0,Y 281.231,Z 664.511,A -85,B 0,C 180,E1 -17388.604,E2 -17388.604} C_VEL
LIN {X 0,Y 281.884,Z 660.926,A -85,B 0,C 180,E1 -17389.29,E2 -17389.29} C_VEL
LIN {X 0,Y 284.701,Z 652.54,A -85,B 0,C 180,E1 -17391.353,E2 -17391.353} C_VEL
LIN {X 0,Y 288.084,Z 642.362,A -85,B 0,C 180,E1 -17393.355,E2 -17393.355} C_VEL
LIN {X 0,Y 291.68,Z 631.059,A -85,B 0,C 180,E1 -17395.13,E2 -17395.13} C_VEL
LIN {X 0,Y 295.422,Z 618.441,A -85,B 0,C 180,E1 -17396.682,E2 -17396.682} C_VEL
LIN {X 0,Y 298.715,Z 606.027,A -85,B 0,C 180,E1 -17397.879,E2 -17397.879} C_VEL
LIN {X 0,Y 302.039,Z 591.42,A -85,B 0,C 180,E1 -17398.965,E2 -17398.965} C_VEL
LIN {X 0,Y 304.872,Z 575.696,A -85,B 0,C 180,E1 -17399.806,E2 -17399.806} C_VEL
LIN {X 0,Y 309.741,Z 536.172,A -85,B 0,C 180,E1 -17401.505,E2 -17401.505} C_VEL
LIN {X 0,Y 310.037,Z 524.664,A -85,B 0,C 180,E1 -17402.328,E2 -17402.328} C_VEL
LIN {X 0,Y 309.758,Z 512.178,A -85,B 0,C 180,E1 -17403.465,E2 -17403.465} C_VEL
LIN {X 0,Y 308.942,Z 499.58,A -85,B 0,C 180,E1 -17404.914,E2 -17404.914} C_VEL
LIN {X 0,Y 307.683,Z 495.922,A -85,B 0,C 180,E1 -17405.77,E2 -17405.77} C_VEL
LIN {X 0,Y 306.153,Z 491.343,A -85,B 0,C 180,E1 -17406.955,E2 -17406.955} C_VEL
LIN {X 0,Y 303.556,Z 484.467,A -85,B 0,C 180,E1 -17409.308,E2 -17409.308} C_VEL
LIN {X 0,Y 301.588,Z 479.937,A -85,B 0,C 180,E1 -17411.78,E2 -17411.78} C_VEL
LIN {X 0,Y 300.736,Z 477.214,A -85,B 0,C 180,E1 -17413.855,E2 -17413.855} C_VEL
LIN {X 0,Y 300.59,Z 475.574,A -85,B 0,C 180,E1 -17415.965,E2 -17415.965} C_VEL
LIN {X 0,Y 301.259,Z 475.019,A -85,B 0,C 180,E1 -17418.29,E2 -17418.29} C_VEL
LIN {X 0,Y 302.606,Z 475.226,A -85,B 0,C 180,E1 -17420.256,E2 -17420.256} C_VEL
LIN {X 0,Y 305.268,Z 477.833,A -85,B 0,C 180,E1 -17422.907,E2 -17422.907} C_VEL
LIN {X 0,Y 308.155,Z 481.219,A -85,B 0,C 180,E1 -17424.948,E2 -17424.948} C_VEL
LIN {X 0,Y 310.469,Z 484.487,A -85,B 0,C 180,E1 -17426.314,E2 -17426.314} C_VEL
LIN {X 0,Y 313.269,Z 488.636,A -85,B 0,C 180,E1 -17427.747,E2 -17427.747} C_VEL
LIN {X 0,Y 314.553,Z 491.129,A -85,B 0,C 180,E1 -17428.391,E2 -17428.391} C_VEL
LIN {X 0,Y 308.292,Z 536.743,A -85,B 0,C 180,E1 -17430.34,E2 -17430.34} C_VEL
LIN {X 0,Y 306.529,Z 550.945,A -85,B 0,C 180,E1 -17431.101,E2 -17431.101} C_VEL
LIN {X 0,Y 304.33,Z 564.803,A -85,B 0,C 180,E1 -17432.145,E2 -17432.145} C_VEL
LIN {X 0,Y 301.757,Z 577.123,A -85,B 0,C 180,E1 -17433.363,E2 -17433.363} C_VEL
LIN {X 0,Y 298.881,Z 588.583,A -85,B 0,C 180,E1 -17434.773,E2 -17434.773} C_VEL
LIN {X 0,Y 295.626,Z 599.803,A -85,B 0,C 180,E1 -17436.534,E2 -17436.534} C_VEL
LIN {X 0,Y 292.866,Z 608.11,A -85,B 0,C 180,E1 -17438.163,E2 -17438.163} C_VEL
LIN {X 0,Y 289.878,Z 616.338,A -85,B 0,C 180,E1 -17440.158,E2 -17440.158} C_VEL
LIN {X 0,Y 287.189,Z 622.975,A -85,B 0,C 180,E1 -17442.188,E2 -17442.188} C_VEL
LIN {X 0,Y 284.683,Z 628.463,A -85,B 0,C 180,E1 -17444.324,E2 -17444.324} C_VEL
LIN {X 0,Y 282.698,Z 632.437,A -85,B 0,C 180,E1 -17446.339,E2 -17446.339} C_VEL
LIN {X 0,Y 280.803,Z 635.514,A -85,B 0,C 180,E1 -17448.45,E2 -17448.45} C_VEL
LIN {X 0,Y 279.722,Z 636.98,A -85,B 0,C 180,E1 -17449.87,E2 -17449.87} C_VEL
LIN {X 0,Y 278.159,Z 638.631,A -85,B 0,C 180,E1 -17452.742,E2 -17452.742} C_VEL
LIN {X 0,Y 277.547,Z 638.84,A -85,B 0,C 180,E1 -17454.187,E2 -17454.187} C_VEL
LIN {X 0,Y 277.016,Z 638.596,A -85,B 0,C 180,E1 -17455.635,E2 -17455.635} C_VEL
LIN {X 0,Y 276.557,Z 637.946,A -85,B 0,C 180,E1 -17457.087,E2 -17457.087} C_VEL
LIN {X 0,Y 276.255,Z 636.886,A -85,B 0,C 180,E1 -17458.542,E2 -17458.542} C_VEL
LIN {X 0,Y 276.103,Z 635.369,A -85,B 0,C 180,E1 -17460,E2 -17460} C_VEL
LIN {X 0,Y 276.088,Z 632.256,A -85,B 0,C 180,E1 -17462.188,E2 -17462.188} C_VEL
LIN {X 0,Y 276.226,Z 628.067,A -85,B 0,C 180,E1 -17464.378,E2 -17464.378} C_VEL
LIN {X 0,Y 276.426,Z 622.686,A -85,B 0,C 180,E1 -17466.57,E2 -17466.57} C_VEL
LIN {X 0,Y 276.788,Z 615.961,A -85,B 0,C 180,E1 -17468.763,E2 -17468.763} C_VEL
LIN {X 0,Y 277.381,Z 607.653,A -85,B 0,C 180,E1 -17470.954,E2 -17470.954} C_VEL
LIN {X 0,Y 278.064,Z 599.171,A -85,B 0,C 180,E1 -17472.777,E2 -17472.777} C_VEL
LIN {X 0,Y 279.014,Z 587.76,A -85,B 0,C 180,E1 -17474.776,E2 -17474.776} C_VEL
LIN {X 0,Y 279.817,Z 576.044,A -85,B 0,C 180,E1 -17476.413,E2 -17476.413} C_VEL
LIN {X 0,Y 280.764,Z 563.219,A -85,B 0,C 180,E1 -17477.841,E2 -17477.841} C_VEL
LIN {X 0,Y 281.427,Z 549.144,A -85,B 0,C 180,E1 -17479.039,E2 -17479.039} C_VEL
LIN {X 0,Y 282.067,Z 536.109,A -85,B 0,C 180,E1 -17479.845,E2 -17479.845} C_VEL
LIN {X 0,Y 282.665,Z 514.046,A -85,B 0,C 180,E1 -17480.751,E2 -17480.751} C_VEL
LIN {X 0,Y 284.521,Z 462.396,A -85,B 0,C 180,E1 -17482.715,E2 -17482.715} C_VEL
LIN {X 0,Y 277.33,Z 439.094,A -85,B 0,C 180,E1 -17483.953,E2 -17483.953} C_VEL
LIN {X 0,Y 277.322,Z 438.932,A -85,B 0,C 180,E1 -17487.503,E2 -17487.503} C_VEL
LIN {X 0,Y 277.274,Z 438.946,A -85,B 0,C 180,E1 -17490.481,E2 -17490.481} C_VEL
LIN {X 0,Y 277.249,Z 438.918,A -85,B 0,C 180,E1 -17493.896,E2 -17493.896} C_VEL
LIN {X 0,Y 277.275,Z 438.95,A -85,B 0,C 180,E1 -17497.468,E2 -17497.468} C_VEL
LIN {X 0,Y 277.211,Z 438.937,A -85,B 0,C 180,E1 -17501.237,E2 -17501.237} C_VEL
LIN {X 0,Y 277.202,Z 438.941,A -85,B 0,C 180,E1 -17505.227,E2 -17505.227} C_VEL
LIN {X 0,Y 277.224,Z 438.942,A -85,B 0,C 180,E1 -17509.512,E2 -17509.512} C_VEL
LIN {X 0,Y 277.291,Z 438.971,A -85,B 0,C 180,E1 -17512.257,E2 -17512.257} C_VEL
LIN {X 0,Y 280.872,Z 450.985,A -85,B 0,C 180,E1 -17515.663,E2 -17515.663} C_VEL
LIN {X 0,Y 284.133,Z 463.939,A -85,B 0,C 180,E1 -17519.05,E2 -17519.05} C_VEL
LIN {X 0,Y 286.206,Z 474.197,A -85,B 0,C 180,E1 -17521.493,E2 -17521.493} C_VEL
LIN {X 0,Y 290.426,Z 496.39,A -85,B 0,C 180,E1 -17522.557,E2 -17522.557} C_VEL
LIN {X 0,Y 292.428,Z 509.472,A -85,B 0,C 180,E1 -17523.116,E2 -17523.116} C_VEL
LIN {X 0,Y 290.5,Z 579.03,A -85,B 0,C 180,E1 -17524.809,E2 -17524.809} C_VEL
LIN {X 0,Y 289.833,Z 592.66,A -85,B 0,C 180,E1 -17525.273,E2 -17525.273} C_VEL
LIN {X 0,Y 288.822,Z 604.777,A -85,B 0,C 180,E1 -17525.947,E2 -17525.947} C_VEL
LIN {X 0,Y 287.5,Z 617.684,A -85,B 0,C 180,E1 -17526.975,E2 -17526.975} C_VEL
LIN {X 0,Y 285.932,Z 629.088,A -85,B 0,C 180,E1 -17528.176,E2 -17528.176} C_VEL
LIN {X 0,Y 284.133,Z 640.496,A -85,B 0,C 180,E1 -17529.739,E2 -17529.739} C_VEL
LIN {X 0,Y 282.453,Z 650.664,A -85,B 0,C 180,E1 -17531.503,E2 -17531.503} C_VEL
LIN {X 0,Y 280.526,Z 660.36,A -85,B 0,C 180,E1 -17533.63,E2 -17533.63} C_VEL
LIN {X 0,Y 278.914,Z 668.149,A -85,B 0,C 180,E1 -17535.778,E2 -17535.778} C_VEL
LIN {X 0,Y 277.88,Z 673.406,A -85,B 0,C 180,E1 -17537.586,E2 -17537.586} C_VEL
LIN {X 0,Y 276.853,Z 678.543,A -85,B 0,C 180,E1 -17539.764,E2 -17539.764} C_VEL
LIN {X 0,Y 276.17,Z 682.517,A -85,B 0,C 180,E1 -17541.954,E2 -17541.954} C_VEL
LIN {X 0,Y 275.708,Z 685.446,A -85,B 0,C 180,E1 -17544.148,E2 -17544.148} C_VEL
LIN {X 0,Y 275.537,Z 686.864,A -85,B 0,C 180,E1 -17545.611,E2 -17545.611} C_VEL
LIN {X 0,Y 275.413,Z 687.858,A -85,B 0,C 180,E1 -17547.075,E2 -17547.075} C_VEL
LIN {X 0,Y 275.273,Z 688.704,A -85,B 0,C 180,E1 -17550,E2 -17550} C_VEL
LIN {X 0,Y 275.301,Z 688.509,A -85,B 0,C 180,E1 -17551.463,E2 -17551.463} C_VEL
LIN {X 0,Y 275.413,Z 687.92,A -85,B 0,C 180,E1 -17552.925,E2 -17552.925} C_VEL
LIN {X 0,Y 275.537,Z 686.95,A -85,B 0,C 180,E1 -17554.389,E2 -17554.389} C_VEL
LIN {X 0,Y 275.783,Z 684.995,A -85,B 0,C 180,E1 -17556.346,E2 -17556.346} C_VEL
LIN {X 0,Y 276.328,Z 681.497,A -85,B 0,C 180,E1 -17558.778,E2 -17558.778} C_VEL
LIN {X 0,Y 277.118,Z 677.216,A -85,B 0,C 180,E1 -17560.965,E2 -17560.965} C_VEL
LIN {X 0,Y 278.256,Z 671.743,A -85,B 0,C 180,E1 -17563.139,E2 -17563.139} C_VEL
LIN {X 0,Y 279.624,Z 664.878,A -85,B 0,C 180,E1 -17565.302,E2 -17565.302} C_VEL
LIN {X 0,Y 281.418,Z 656.287,A -85,B 0,C 180,E1 -17567.439,E2 -17567.439} C_VEL
LIN {X 0,Y 283.051,Z 647.216,A -85,B 0,C 180,E1 -17569.26,E2 -17569.26} C_VEL
LIN {X 0,Y 284.805,Z 636.533,A -85,B 0,C 180,E1 -17570.966,E2 -17570.966} C_VEL
LIN {X 0,Y 286.471,Z 625.508,A -85,B 0,C 180,E1 -17572.35,E2 -17572.35} C_VEL
LIN {X 0,Y 287.93,Z 614.122,A -85,B 0,C 180,E1 -17573.464,E2 -17573.464} C_VEL
LIN {X 0,Y 289.26,Z 601.06,A -85,B 0,C 180,E1 -17574.396,E2 -17574.396} C_VEL
LIN {X 0,Y 290.014,Z 589.072,A -85,B 0,C 180,E1 -17574.997,E2 -17574.997} C_VEL
LIN {X 0,Y 290.732,Z 572.811,A -85,B 0,C 180,E1 -17575.457,E2 -17575.457} C_VEL
LIN {X 0,Y 292.432,Z 508.314,A -85,B 0,C 180,E1 -17577.035,E2 -17577.035} C_VEL
LIN {X 0,Y 287.605,Z 480.868,A -85,B 0,C 180,E1 -17578.291,E2 -17578.291} C_VEL
LIN {X 0,Y 286.219,Z 474.066,A -85,B 0,C 180,E1 -17578.66,E2 -17578.66} C_VEL
LIN {X 0,Y 283.921,Z 462.953,A -85,B 0,C 180,E1 -17581.32,E2 -17581.32} C_VEL
LIN {X 0,Y 280.979,Z 451.388,A -85,B 0,C 180,E1 -17584.369,E2 -17584.369} C_VEL
LIN {X 0,Y 277.748,Z 440.644,A -85,B 0,C 180,E1 -17587.394,E2 -17587.394} C_VEL
LIN {X 0,Y 277.284,Z 438.942,A -85,B 0,C 180,E1 -17587.961,E2 -17587.961} C_VEL
LIN {X 0,Y 277.218,Z 438.948,A -85,B 0,C 180,E1 -17592.25,E2 -17592.25} C_VEL
LIN {X 0,Y 276.574,Z 439.034,A -85,B 0,C 180,E1 -17593.463,E2 -17593.463} C_VEL
LIN {X 0,Y 273.695,Z 439.395,A -85,B 0,C 180,E1 -17595.437,E2 -17595.437} C_VEL
LIN {X 0,Y 271.25,Z 439.691,A -85,B 0,C 180,E1 -17597.042,E2 -17597.042} C_VEL
LIN {X 0,Y 270.227,Z 439.811,A -85,B 0,C 180,E1 -17598.287,E2 -17598.287} C_VEL
LIN {X 0,Y 270.158,Z 439.82,A -85,B 0,C 180,E1 -17598.709,E2 -17598.709} C_VEL
LIN {X 0,Y 270.209,Z 439.827,A -85,B 0,C 180,E1 -17601.374,E2 -17601.374} C_VEL
LIN {X 0,Y 270.206,Z 439.817,A -85,B 0,C 180,E1 -17605.095,E2 -17605.095} C_VEL
LIN {X 0,Y 270.267,Z 439.856,A -85,B 0,C 180,E1 -17607.068,E2 -17607.068} C_VEL
LIN {X 0,Y 274.06,Z 457.742,A -85,B 0,C 180,E1 -17611.407,E2 -17611.407} C_VEL
LIN {X 0,Y 275.311,Z 464.816,A -85,B 0,C 180,E1 -17613.069,E2 -17613.069} C_VEL
LIN {X 0,Y 274.666,Z 473.708,A -85,B 0,C 180,E1 -17615.027,E2 -17615.027} C_VEL
LIN {X 0,Y 274.536,Z 475.242,A -85,B 0,C 180,E1 -17615.317,E2 -17615.317} C_VEL
LIN {X 0,Y 277.336,Z 502.057,A -85,B 0,C 180,E1 -17616.535,E2 -17616.535} C_VEL
LIN {X 0,Y 277.845,Z 506.449,A -85,B 0,C 180,E1 -17616.733,E2 -17616.733} C_VEL
LIN {X 0,Y 274.764,Z 586.433,A -85,B 0,C 180,E1 -17619.897,E2 -17619.897} C_VEL
LIN {X 0,Y 274.092,Z 600.192,A -85,B 0,C 180,E1 -17620.723,E2 -17620.723} C_VEL
LIN {X 0,Y 273.181,Z 613.477,A -85,B 0,C 180,E1 -17621.824,E2 -17621.824} C_VEL
LIN {X 0,Y 272.355,Z 624.866,A -85,B 0,C 180,E1 -17623.044,E2 -17623.044} C_VEL
LIN {X 0,Y 271.581,Z 635.323,A -85,B 0,C 180,E1 -17624.426,E2 -17624.426} C_VEL
LIN {X 0,Y 270.606,Z 646.652,A -85,B 0,C 180,E1 -17626.291,E2 -17626.291} C_VEL
LIN {X 0,Y 269.741,Z 656.715,A -85,B 0,C 180,E1 -17628.35,E2 -17628.35} C_VEL
LIN {X 0,Y 269.072,Z 665.598,A -85,B 0,C 180,E1 -17630.605,E2 -17630.605} C_VEL
LIN {X 0,Y 268.585,Z 672.682,A -85,B 0,C 180,E1 -17632.86,E2 -17632.86} C_VEL
LIN {X 0,Y 268.302,Z 679.181,A -85,B 0,C 180,E1 -17635.493,E2 -17635.493} C_VEL
LIN {X 0,Y 268.249,Z 683.359,A -85,B 0,C 180,E1 -17637.748,E2 -17637.748} C_VEL
LIN {X 0,Y 268.191,Z 686.403,A -85,B 0,C 180,E1 -17640,E2 -17640} C_VEL
LIN {X 0,Y 268.248,Z 687.839,A -85,B 0,C 180,E1 -17641.501,E2 -17641.501} C_VEL
LIN {X 0,Y 268.348,Z 688.867,A -85,B 0,C 180,E1 -17643.002,E2 -17643.002} C_VEL
LIN {X 0,Y 268.56,Z 689.445,A -85,B 0,C 180,E1 -17644.503,E2 -17644.503} C_VEL
LIN {X 0,Y 269.213,Z 689.392,A -85,B 0,C 180,E1 -17647.243,E2 -17647.243} C_VEL
LIN {X 0,Y 269.818,Z 688.645,A -85,B 0,C 180,E1 -17648.991,E2 -17648.991} C_VEL
LIN {X 0,Y 270.562,Z 687.518,A -85,B 0,C 180,E1 -17650.476,E2 -17650.476} C_VEL
LIN {X 0,Y 271.465,Z 685.981,A -85,B 0,C 180,E1 -17651.953,E2 -17651.953} C_VEL
LIN {X 0,Y 272.994,Z 682.839,A -85,B 0,C 180,E1 -17654.156,E2 -17654.156} C_VEL
LIN {X 0,Y 275.065,Z 678.63,A -85,B 0,C 180,E1 -17656.323,E2 -17656.323} C_VEL
LIN {X 0,Y 277.903,Z 672.246,A -85,B 0,C 180,E1 -17658.811,E2 -17658.811} C_VEL
LIN {X 0,Y 280.795,Z 665.283,A -85,B 0,C 180,E1 -17660.895,E2 -17660.895} C_VEL
LIN {X 0,Y 284.086,Z 656.825,A -85,B 0,C 180,E1 -17662.932,E2 -17662.932} C_VEL
LIN {X 0,Y 287.619,Z 646.677,A -85,B 0,C 180,E1 -17664.862,E2 -17664.862} C_VEL
LIN {X 0,Y 291.427,Z 634.459,A -85,B 0,C 180,E1 -17666.69,E2 -17666.69} C_VEL
LIN {X 0,Y 294.59,Z 622.89,A -85,B 0,C 180,E1 -17668.041,E2 -17668.041} C_VEL
LIN {X 0,Y 297.437,Z 610.621,A -85,B 0,C 180,E1 -17669.166,E2 -17669.166} C_VEL
LIN {X 0,Y 300.172,Z 596.645,A -85,B 0,C 180,E1 -17670.127,E2 -17670.127} C_VEL
LIN {X 0,Y 302.682,Z 580.072,A -85,B 0,C 180,E1 -17670.912,E2 -17670.912} C_VEL
LIN {X 0,Y 311.133,Z 521.012,A -85,B 0,C 180,E1 -17673.469,E2 -17673.469} C_VEL
LIN {X 0,Y 310.705,Z 512.307,A -85,B 0,C 180,E1 -17674.509,E2 -17674.509} C_VEL
LIN {X 0,Y 308.601,Z 506.209,A -85,B 0,C 180,E1 -17676.095,E2 -17676.095} C_VEL
LIN {X 0,Y 306.99,Z 502.128,A -85,B 0,C 180,E1 -17677.471,E2 -17677.471} C_VEL
LIN {X 0,Y 305.203,Z 497.9,A -85,B 0,C 180,E1 -17679.36,E2 -17679.36} C_VEL
LIN {X 0,Y 303.653,Z 494.466,A -85,B 0,C 180,E1 -17681.777,E2 -17681.777} C_VEL
LIN {X 0,Y 303.15,Z 493.047,A -85,B 0,C 180,E1 -17683.432,E2 -17683.432} C_VEL
LIN {X 0,Y 303.174,Z 492.334,A -85,B 0,C 180,E1 -17685.941,E2 -17685.941} C_VEL
LIN {X 0,Y 304.265,Z 493.043,A -85,B 0,C 180,E1 -17688.427,E2 -17688.427} C_VEL
LIN {X 0,Y 306.713,Z 495.467,A -85,B 0,C 180,E1 -17691.176,E2 -17691.176} C_VEL
LIN {X 0,Y 308.727,Z 498.478,A -85,B 0,C 180,E1 -17692.864,E2 -17692.864} C_VEL
LIN {X 0,Y 309.424,Z 502.912,A -85,B 0,C 180,E1 -17693.804,E2 -17693.804} C_VEL
LIN {X 0,Y 309.338,Z 516.769,A -85,B 0,C 180,E1 -17695.343,E2 -17695.343} C_VEL
LIN {X 0,Y 308.869,Z 530.334,A -85,B 0,C 180,E1 -17696.556,E2 -17696.556} C_VEL
LIN {X 0,Y 307.862,Z 541.602,A -85,B 0,C 180,E1 -17697.299,E2 -17697.299} C_VEL
LIN {X 0,Y 298.603,Z 605.453,A -85,B 0,C 180,E1 -17700.136,E2 -17700.136} C_VEL
LIN {X 0,Y 296.158,Z 617.941,A -85,B 0,C 180,E1 -17700.891,E2 -17700.891} C_VEL
LIN {X 0,Y 292.723,Z 632.271,A -85,B 0,C 180,E1 -17702.084,E2 -17702.084} C_VEL
LIN {X 0,Y 288.879,Z 646.121,A -85,B 0,C 180,E1 -17703.641,E2 -17703.641} C_VEL
LIN {X 0,Y 285.351,Z 657.179,A -85,B 0,C 180,E1 -17705.247,E2 -17705.247} C_VEL
LIN {X 0,Y 281.675,Z 667.961,A -85,B 0,C 180,E1 -17707.248,E2 -17707.248} C_VEL
LIN {X 0,Y 278.498,Z 676.75,A -85,B 0,C 180,E1 -17709.311,E2 -17709.311} C_VEL
LIN {X 0,Y 275.686,Z 683.913,A -85,B 0,C 180,E1 -17711.418,E2 -17711.418} C_VEL
LIN {X 0,Y 273.329,Z 689.731,A -85,B 0,C 180,E1 -17713.57,E2 -17713.57} C_VEL
LIN {X 0,Y 271.616,Z 694.313,A -85,B 0,C 180,E1 -17715.77,E2 -17715.77} C_VEL
LIN {X 0,Y 270.17,Z 697.845,A -85,B 0,C 180,E1 -17717.989,E2 -17717.989} C_VEL
LIN {X 0,Y 269.478,Z 699.631,A -85,B 0,C 180,E1 -17719.481,E2 -17719.481} C_VEL
LIN {X 0,Y 268.96,Z 701,A -85,B 0,C 180,E1 -17720.98,E2 -17720.98} C_VEL
LIN {X 0,Y 268.551,Z 701.908,A -85,B 0,C 180,E1 -17722.481,E2 -17722.481} C_VEL
LIN {X 0,Y 268.261,Z 702.494,A -85,B 0,C 180,E1 -17724.587,E2 -17724.587} C_VEL
LIN {X 0,Y 268.266,Z 702.35,A -85,B 0,C 180,E1 -17726.997,E2 -17726.997} C_VEL
LIN {X 0,Y 268.237,Z 702.964,A -85,B 0,C 180,E1 -17728.499,E2 -17728.499} C_VEL
LIN {X 0,Y 268.251,Z 703.182,A -85,B 0,C 180,E1 -17730,E2 -17730} C_VEL
LIN {X 0,Y 268.229,Z 702.955,A -85,B 0,C 180,E1 -17731.501,E2 -17731.501} C_VEL
LIN {X 0,Y 268.224,Z 702.334,A -85,B 0,C 180,E1 -17733.004,E2 -17733.004} C_VEL
LIN {X 0,Y 268.236,Z 700.545,A -85,B 0,C 180,E1 -17735.357,E2 -17735.357} C_VEL
LIN {X 0,Y 268.589,Z 696.897,A -85,B 0,C 180,E1 -17738.274,E2 -17738.274} C_VEL
LIN {X 0,Y 269.162,Z 692.849,A -85,B 0,C 180,E1 -17740.531,E2 -17740.531} C_VEL
LIN {X 0,Y 270.169,Z 686.609,A -85,B 0,C 180,E1 -17743.157,E2 -17743.157} C_VEL
LIN {X 0,Y 271.617,Z 679.812,A -85,B 0,C 180,E1 -17745.38,E2 -17745.38} C_VEL
LIN {X 0,Y 272.97,Z 672.853,A -85,B 0,C 180,E1 -17747.223,E2 -17747.223} C_VEL
LIN {X 0,Y 274.798,Z 662.819,A -85,B 0,C 180,E1 -17749.419,E2 -17749.419} C_VEL
LIN {X 0,Y 277.635,Z 655.059,A -85,B 0,C 180,E1 -17751.534,E2 -17751.534} C_VEL
LIN {X 0,Y 281.056,Z 645.689,A -85,B 0,C 180,E1 -17753.584,E2 -17753.584} C_VEL
LIN {X 0,Y 285.065,Z 634.319,A -85,B 0,C 180,E1 -17755.559,E2 -17755.559} C_VEL
LIN {X 0,Y 289.246,Z 621.502,A -85,B 0,C 180,E1 -17757.298,E2 -17757.298} C_VEL
LIN {X 0,Y 293.088,Z 608.456,A -85,B 0,C 180,E1 -17758.658,E2 -17758.658} C_VEL
LIN {X 0,Y 296.608,Z 594.936,A -85,B 0,C 180,E1 -17759.743,E2 -17759.743} C_VEL
LIN {X 0,Y 299.748,Z 579.817,A -85,B 0,C 180,E1 -17760.661,E2 -17760.661} C_VEL
LIN {X 0,Y 303.224,Z 555.12,A -85,B 0,C 180,E1 -17761.774,E2 -17761.774} C_VEL
LIN {X 0,Y 305.577,Z 537.277,A -85,B 0,C 180,E1 -17762.566,E2 -17762.566} C_VEL
LIN {X 0,Y 306.009,Z 526.514,A -85,B 0,C 180,E1 -17763.368,E2 -17763.368} C_VEL
LIN {X 0,Y 305.968,Z 515.294,A -85,B 0,C 180,E1 -17764.424,E2 -17764.424} C_VEL
LIN {X 0,Y 305.524,Z 503.984,A -85,B 0,C 180,E1 -17765.755,E2 -17765.755} C_VEL
LIN {X 0,Y 303.337,Z 497.079,A -85,B 0,C 180,E1 -17767.558,E2 -17767.558} C_VEL
LIN {X 0,Y 301.163,Z 490.61,A -85,B 0,C 180,E1 -17769.826,E2 -17769.826} C_VEL
LIN {X 0,Y 299.414,Z 485.934,A -85,B 0,C 180,E1 -17772.468,E2 -17772.468} C_VEL
LIN {X 0,Y 298.807,Z 483.331,A -85,B 0,C 180,E1 -17774.719,E2 -17774.719} C_VEL
LIN {X 0,Y 299.004,Z 482.076,A -85,B 0,C 180,E1 -17777.028,E2 -17777.028} C_VEL
LIN {X 0,Y 300.531,Z 481.912,A -85,B 0,C 180,E1 -17779.883,E2 -17779.883} C_VEL
LIN {X 0,Y 303.137,Z 484.487,A -85,B 0,C 180,E1 -17782.668,E2 -17782.668} C_VEL
LIN {X 0,Y 305.799,Z 487.743,A -85,B 0,C 180,E1 -17784.657,E2 -17784.657} C_VEL
LIN {X 0,Y 308.95,Z 492.327,A -85,B 0,C 180,E1 -17786.565,E2 -17786.565} C_VEL
LIN {X 0,Y 310.493,Z 495.017,A -85,B 0,C 180,E1 -17787.406,E2 -17787.406} C_VEL
LIN {X 0,Y 304.187,Z 537.9,A -85,B 0,C 180,E1 -17789.279,E2 -17789.279} C_VEL
LIN {X 0,Y 302.235,Z 552.384,A -85,B 0,C 180,E1 -17790.075,E2 -17790.075} C_VEL
LIN {X 0,Y 299.867,Z 565.627,A -85,B 0,C 180,E1 -17791.093,E2 -17791.093} C_VEL
LIN {X 0,Y 296.76,Z 579.51,A -85,B 0,C 180,E1 -17792.496,E2 -17792.496} C_VEL
LIN {X 0,Y 293.71,Z 590.562,A -85,B 0,C 180,E1 -17793.916,E2 -17793.916} C_VEL
LIN {X 0,Y 290.249,Z 601.465,A -85,B 0,C 180,E1 -17795.693,E2 -17795.693} C_VEL
LIN {X 0,Y 287.295,Z 609.672,A -85,B 0,C 180,E1 -17797.338,E2 -17797.338} C_VEL
LIN {X 0,Y 284.08,Z 617.689,A -85,B 0,C 180,E1 -17799.357,E2 -17799.357} C_VEL
LIN {X 0,Y 280.759,Z 625.177,A -85,B 0,C 180,E1 -17801.766,E2 -17801.766} C_VEL
LIN {X 0,Y 278.175,Z 630.2,A -85,B 0,C 180,E1 -17803.864,E2 -17803.864} C_VEL
LIN {X 0,Y 275.98,Z 634.043,A -85,B 0,C 180,E1 -17806,E2 -17806} C_VEL
LIN {X 0,Y 273.986,Z 636.906,A -85,B 0,C 180,E1 -17808.158,E2 -17808.158} C_VEL
LIN {X 0,Y 272.848,Z 638.244,A -85,B 0,C 180,E1 -17809.612,E2 -17809.612} C_VEL
LIN {X 0,Y 271.933,Z 639.153,A -85,B 0,C 180,E1 -17811.079,E2 -17811.079} C_VEL
LIN {X 0,Y 271.194,Z 639.619,A -85,B 0,C 180,E1 -17812.555,E2 -17812.555} C_VEL
LIN {X 0,Y 270.554,Z 639.659,A -85,B 0,C 180,E1 -17814.036,E2 -17814.036} C_VEL
LIN {X 0,Y 269.985,Z 639.308,A -85,B 0,C 180,E1 -17815.521,E2 -17815.521} C_VEL
LIN {X 0,Y 269.501,Z 638.549,A -85,B 0,C 180,E1 -17817.01,E2 -17817.01} C_VEL
LIN {X 0,Y 269.194,Z 637.324,A -85,B 0,C 180,E1 -17818.504,E2 -17818.504} C_VEL
LIN {X 0,Y 268.994,Z 634.696,A -85,B 0,C 180,E1 -17820.749,E2 -17820.749} C_VEL
LIN {X 0,Y 268.989,Z 631.047,A -85,B 0,C 180,E1 -17822.995,E2 -17822.995} C_VEL
LIN {X 0,Y 269.264,Z 626.256,A -85,B 0,C 180,E1 -17825.242,E2 -17825.242} C_VEL
LIN {X 0,Y 269.461,Z 619.727,A -85,B 0,C 180,E1 -17827.646,E2 -17827.646} C_VEL
LIN {X 0,Y 269.896,Z 612.664,A -85,B 0,C 180,E1 -17829.745,E2 -17829.745} C_VEL
LIN {X 0,Y 270.648,Z 603.334,A -85,B 0,C 180,E1 -17831.99,E2 -17831.99} C_VEL
LIN {X 0,Y 271.487,Z 592.801,A -85,B 0,C 180,E1 -17834.046,E2 -17834.046} C_VEL
LIN {X 0,Y 272.359,Z 582.184,A -85,B 0,C 180,E1 -17835.721,E2 -17835.721} C_VEL
LIN {X 0,Y 273.233,Z 570.651,A -85,B 0,C 180,E1 -17837.206,E2 -17837.206} C_VEL
LIN {X 0,Y 273.981,Z 557.67,A -85,B 0,C 180,E1 -17838.527,E2 -17838.527} C_VEL
LIN {X 0,Y 274.706,Z 543.309,A -85,B 0,C 180,E1 -17839.621,E2 -17839.621} C_VEL
LIN {X 0,Y 275.172,Z 530.247,A -85,B 0,C 180,E1 -17840.316,E2 -17840.316} C_VEL
LIN {X 0,Y 277.524,Z 463.701,A -85,B 0,C 180,E1 -17842.936,E2 -17842.936} C_VEL
LIN {X 0,Y 270.269,Z 439.815,A -85,B 0,C 180,E1 -17844.278,E2 -17844.278} C_VEL
LIN {X 0,Y 270.271,Z 439.81,A -85,B 0,C 180,E1 -17847.909,E2 -17847.909} C_VEL
LIN {X 0,Y 270.186,Z 439.821,A -85,B 0,C 180,E1 -17851.348,E2 -17851.348} C_VEL
LIN {X 0,Y 270.204,Z 439.802,A -85,B 0,C 180,E1 -17854.905,E2 -17854.905} C_VEL
LIN {X 0,Y 270.199,Z 439.821,A -85,B 0,C 180,E1 -17858.71,E2 -17858.71} C_VEL
LIN {X 0,Y 270.174,Z 439.831,A -85,B 0,C 180,E1 -17862.558,E2 -17862.558} C_VEL
LIN {X 0,Y 270.167,Z 439.819,A -85,B 0,C 180,E1 -17866.751,E2 -17866.751} C_VEL
LIN {X 0,Y 270.224,Z 439.823,A -85,B 0,C 180,E1 -17871.283,E2 -17871.283} C_VEL
LIN {X 0,Y 270.302,Z 440.376,A -85,B 0,C 180,E1 -17871.531,E2 -17871.531} C_VEL
LIN {X 0,Y 273.127,Z 449.223,A -85,B 0,C 180,E1 -17874.149,E2 -17874.149} C_VEL
LIN {X 0,Y 276.354,Z 461.242,A -85,B 0,C 180,E1 -17877.45,E2 -17877.45} C_VEL
LIN {X 0,Y 278.673,Z 471.408,A -85,B 0,C 180,E1 -17880.023,E2 -17880.023} C_VEL
LIN {X 0,Y 279.323,Z 474.623,A -85,B 0,C 180,E1 -17880.733,E2 -17880.733} C_VEL
LIN {X 0,Y 280.787,Z 478.867,A -85,B 0,C 180,E1 -17881.023,E2 -17881.023} C_VEL
LIN {X 0,Y 285.572,Z 506.109,A -85,B 0,C 180,E1 -17882.32,E2 -17882.32} C_VEL
LIN {X 0,Y 286.1,Z 510.535,A -85,B 0,C 180,E1 -17882.499,E2 -17882.499} C_VEL
LIN {X 0,Y 284.107,Z 579.135,A -85,B 0,C 180,E1 -17884.201,E2 -17884.201} C_VEL
LIN {X 0,Y 283.418,Z 592.808,A -85,B 0,C 180,E1 -17884.675,E2 -17884.675} C_VEL
LIN {X 0,Y 282.351,Z 604.943,A -85,B 0,C 180,E1 -17885.359,E2 -17885.359} C_VEL
LIN {X 0,Y 280.999,Z 617.858,A -85,B 0,C 180,E1 -17886.411,E2 -17886.411} C_VEL
LIN {X 0,Y 279.345,Z 629.268,A -85,B 0,C 180,E1 -17887.633,E2 -17887.633} C_VEL
LIN {X 0,Y 277.48,Z 640.68,A -85,B 0,C 180,E1 -17889.231,E2 -17889.231} C_VEL
LIN {X 0,Y 275.719,Z 650.85,A -85,B 0,C 180,E1 -17891.035,E2 -17891.035} C_VEL
LIN {X 0,Y 273.727,Z 660.547,A -85,B 0,C 180,E1 -17893.211,E2 -17893.211} C_VEL
LIN {X 0,Y 272.023,Z 668.337,A -85,B 0,C 180,E1 -17895.41,E2 -17895.41} C_VEL
LIN {X 0,Y 270.958,Z 673.595,A -85,B 0,C 180,E1 -17897.263,E2 -17897.263} C_VEL
LIN {X 0,Y 269.853,Z 678.733,A -85,B 0,C 180,E1 -17899.496,E2 -17899.496} C_VEL
LIN {X 0,Y 269.128,Z 682.707,A -85,B 0,C 180,E1 -17901.742,E2 -17901.742} C_VEL
LIN {X 0,Y 268.649,Z 685.635,A -85,B 0,C 180,E1 -17903.993,E2 -17903.993} C_VEL
LIN {X 0,Y 268.467,Z 687.053,A -85,B 0,C 180,E1 -17905.496,E2 -17905.496} C_VEL
LIN {X 0,Y 268.327,Z 688.047,A -85,B 0,C 180,E1 -17906.997,E2 -17906.997} C_VEL
LIN {X 0,Y 268.198,Z 688.893,A -85,B 0,C 180,E1 -17910,E2 -17910} C_VEL
LIN {X 0,Y 268.229,Z 688.697,A -85,B 0,C 180,E1 -17911.501,E2 -17911.501} C_VEL
LIN {X 0,Y 268.327,Z 688.108,A -85,B 0,C 180,E1 -17913.003,E2 -17913.003} C_VEL
LIN {X 0,Y 268.467,Z 687.138,A -85,B 0,C 180,E1 -17914.504,E2 -17914.504} C_VEL
LIN {X 0,Y 268.711,Z 685.379,A -85,B 0,C 180,E1 -17916.344,E2 -17916.344} C_VEL
LIN {X 0,Y 269.297,Z 681.685,A -85,B 0,C 180,E1 -17919.009,E2 -17919.009} C_VEL
LIN {X 0,Y 270.15,Z 677.403,A -85,B 0,C 180,E1 -17921.251,E2 -17921.251} C_VEL
LIN {X 0,Y 271.34,Z 671.929,A -85,B 0,C 180,E1 -17923.48,E2 -17923.48} C_VEL
LIN {X 0,Y 272.758,Z 665.062,A -85,B 0,C 180,E1 -17925.697,E2 -17925.697} C_VEL
LIN {X 0,Y 274.641,Z 656.468,A -85,B 0,C 180,E1 -17927.883,E2 -17927.883} C_VEL
LIN {X 0,Y 276.443,Z 646.904,A -85,B 0,C 180,E1 -17929.838,E2 -17929.838} C_VEL
LIN {X 0,Y 278.195,Z 636.706,A -85,B 0,C 180,E1 -17931.488,E2 -17931.488} C_VEL
LIN {X 0,Y 279.94,Z 625.676,A -85,B 0,C 180,E1 -17932.901,E2 -17932.901} C_VEL
LIN {X 0,Y 281.452,Z 614.281,A -85,B 0,C 180,E1 -17934.037,E2 -17934.037} C_VEL
LIN {X 0,Y 282.808,Z 601.203,A -85,B 0,C 180,E1 -17934.99,E2 -17934.99} C_VEL
LIN {X 0,Y 283.702,Z 588.154,A -85,B 0,C 180,E1 -17935.642,E2 -17935.642} C_VEL
LIN {X 0,Y 284.599,Z 563.961,A -85,B 0,C 180,E1 -17936.293,E2 -17936.293} C_VEL
LIN {X 0,Y 286.159,Z 509.557,A -85,B 0,C 180,E1 -17937.645,E2 -17937.645} C_VEL
LIN {X 0,Y 281.5,Z 482.755,A -85,B 0,C 180,E1 -17938.909,E2 -17938.909} C_VEL
LIN {X 0,Y 280.058,Z 476.459,A -85,B 0,C 180,E1 -17939.255,E2 -17939.255} C_VEL
LIN {X 0,Y 279.247,Z 474.163,A -85,B 0,C 180,E1 -17939.451,E2 -17939.451} C_VEL
LIN {X 0,Y 276.656,Z 462.249,A -85,B 0,C 180,E1 -17942.412,E2 -17942.412} C_VEL
LIN {X 0,Y 273.24,Z 449.587,A -85,B 0,C 180,E1 -17945.884,E2 -17945.884} C_VEL
LIN {X 0,Y 270.206,Z 439.829,A -85,B 0,C 180,E1 -17948.841,E2 -17948.841} C_VEL
LIN {X 0,Y 270.194,Z 439.827,A -85,B 0,C 180,E1 -17952.554,E2 -17952.554} C_VEL
LIN {X 0,Y 270.174,Z 439.829,A -85,B 0,C 180,E1 -17956.749,E2 -17956.749} C_VEL
LIN {X 0,Y 270.158,Z 439.82,A -85,B 0,C 180,E1 -17958.709,E2 -17958.709} C_VEL
LIN {X 0,Y 269.523,Z 439.913,A -85,B 0,C 180,E1 -17959.954,E2 -17959.954} C_VEL
LIN {X 0,Y 266.663,Z 440.26,A -85,B 0,C 180,E1 -17961.983,E2 -17961.983} C_VEL
LIN {X 0,Y 264.231,Z 440.554,A -85,B 0,C 180,E1 -17963.633,E2 -17963.633} C_VEL
LIN {X 0,Y 263.212,Z 440.685,A -85,B 0,C 180,E1 -17964.913,E2 -17964.913} C_VEL
LIN {X 0,Y 263.144,Z 440.696,A -85,B 0,C 180,E1 -17965.346,E2 -17965.346} C_VEL
LIN {X 0,Y 263.232,Z 440.9,A -85,B 0,C 180,E1 -17966.816,E2 -17966.816} C_VEL
LIN {X 0,Y 266.42,Z 455.885,A -85,B 0,C 180,E1 -17970.52,E2 -17970.52} C_VEL
LIN {X 0,Y 268.33,Z 465.915,A -85,B 0,C 180,E1 -17972.938,E2 -17972.938} C_VEL
LIN {X 0,Y 267.566,Z 475.156,A -85,B 0,C 180,E1 -17974.993,E2 -17974.993} C_VEL
LIN {X 0,Y 270.217,Z 501.626,A -85,B 0,C 180,E1 -17976.232,E2 -17976.232} C_VEL
LIN {X 0,Y 270.793,Z 507.692,A -85,B 0,C 180,E1 -17976.509,E2 -17976.509} C_VEL
LIN {X 0,Y 267.716,Z 586.594,A -85,B 0,C 180,E1 -17979.745,E2 -17979.745} C_VEL
LIN {X 0,Y 266.963,Z 601.509,A -85,B 0,C 180,E1 -17980.688,E2 -17980.688} C_VEL
LIN {X 0,Y 266.066,Z 614.128,A -85,B 0,C 180,E1 -17981.792,E2 -17981.792} C_VEL
LIN {X 0,Y 265.068,Z 626.942,A -85,B 0,C 180,E1 -17983.241,E2 -17983.241} C_VEL
LIN {X 0,Y 264.327,Z 636.455,A -85,B 0,C 180,E1 -17984.58,E2 -17984.58} C_VEL
LIN {X 0,Y 263.497,Z 646.61,A -85,B 0,C 180,E1 -17986.307,E2 -17986.307} C_VEL
LIN {X 0,Y 262.641,Z 656.743,A -85,B 0,C 180,E1 -17988.422,E2 -17988.422} C_VEL
LIN {X 0,Y 261.964,Z 665.671,A -85,B 0,C 180,E1 -17990.737,E2 -17990.737} C_VEL
LIN {X 0,Y 261.471,Z 672.799,A -85,B 0,C 180,E1 -17993.053,E2 -17993.053} C_VEL
LIN {X 0,Y 261.215,Z 678.482,A -85,B 0,C 180,E1 -17995.37,E2 -17995.37} C_VEL
LIN {X 0,Y 261.184,Z 682.87,A -85,B 0,C 180,E1 -17997.687,E2 -17997.687} C_VEL
LIN {X 0,Y 261.117,Z 686.118,A -85,B 0,C 180,E1 -18000,E2 -18000} C_VEL
LIN {X 0,Y 261.177,Z 687.706,A -85,B 0,C 180,E1 -18001.542,E2 -18001.542} C_VEL
LIN {X 0,Y 261.267,Z 688.835,A -85,B 0,C 180,E1 -18003.084,E2 -18003.084} C_VEL
LIN {X 0,Y 261.479,Z 689.561,A -85,B 0,C 180,E1 -18004.625,E2 -18004.625} C_VEL
LIN {X 0,Y 262.115,Z 689.812,A -85,B 0,C 180,E1 -18007.219,E2 -18007.219} C_VEL
LIN {X 0,Y 262.835,Z 689.157,A -85,B 0,C 180,E1 -18009.232,E2 -18009.232} C_VEL
LIN {X 0,Y 263.635,Z 688.201,A -85,B 0,C 180,E1 -18010.755,E2 -18010.755} C_VEL
LIN {X 0,Y 265.624,Z 684.965,A -85,B 0,C 180,E1 -18013.776,E2 -18013.776} C_VEL
LIN {X 0,Y 267.567,Z 681.398,A -85,B 0,C 180,E1 -18016.009,E2 -18016.009} C_VEL
LIN {X 0,Y 270.068,Z 676.683,A -85,B 0,C 180,E1 -18018.197,E2 -18018.197} C_VEL
LIN {X 0,Y 273.32,Z 669.727,A -85,B 0,C 180,E1 -18020.705,E2 -18020.705} C_VEL
LIN {X 0,Y 276.675,Z 662.188,A -85,B 0,C 180,E1 -18022.791,E2 -18022.791} C_VEL
LIN {X 0,Y 280.374,Z 652.959,A -85,B 0,C 180,E1 -18024.826,E2 -18024.826} C_VEL
LIN {X 0,Y 283.765,Z 643.683,A -85,B 0,C 180,E1 -18026.475,E2 -18026.475} C_VEL
LIN {X 0,Y 287.422,Z 632.347,A -85,B 0,C 180,E1 -18028.08,E2 -18028.08} C_VEL
LIN {X 0,Y 290.997,Z 619.865,A -85,B 0,C 180,E1 -18029.478,E2 -18029.478} C_VEL
LIN {X 0,Y 293.915,Z 607.709,A -85,B 0,C 180,E1 -18030.524,E2 -18030.524} C_VEL
LIN {X 0,Y 296.294,Z 595.748,A -85,B 0,C 180,E1 -18031.313,E2 -18031.313} C_VEL
LIN {X 0,Y 299.814,Z 573.061,A -85,B 0,C 180,E1 -18032.377,E2 -18032.377} C_VEL
LIN {X 0,Y 307.623,Z 523.396,A -85,B 0,C 180,E1 -18034.532,E2 -18034.532} C_VEL
LIN {X 0,Y 307.393,Z 516.857,A -85,B 0,C 180,E1 -18035.344,E2 -18035.344} C_VEL
LIN {X 0,Y 305.73,Z 511.577,A -85,B 0,C 180,E1 -18036.814,E2 -18036.814} C_VEL
LIN {X 0,Y 304.384,Z 507.782,A -85,B 0,C 180,E1 -18038.163,E2 -18038.163} C_VEL
LIN {X 0,Y 302.993,Z 504.147,A -85,B 0,C 180,E1 -18039.862,E2 -18039.862} C_VEL
LIN {X 0,Y 301.674,Z 500.795,A -85,B 0,C 180,E1 -18042.344,E2 -18042.344} C_VEL
LIN {X 0,Y 301.288,Z 499.505,A -85,B 0,C 180,E1 -18044.411,E2 -18044.411} C_VEL
LIN {X 0,Y 301.531,Z 499.214,A -85,B 0,C 180,E1 -18046.265,E2 -18046.265} C_VEL
LIN {X 0,Y 302.712,Z 500.14,A -85,B 0,C 180,E1 -18048.759,E2 -18048.759} C_VEL
LIN {X 0,Y 305.007,Z 502.534,A -85,B 0,C 180,E1 -18051.257,E2 -18051.257} C_VEL
LIN {X 0,Y 306.155,Z 504.826,A -85,B 0,C 180,E1 -18052.371,E2 -18052.371} C_VEL
LIN {X 0,Y 306.474,Z 507.353,A -85,B 0,C 180,E1 -18052.898,E2 -18052.898} C_VEL
LIN {X 0,Y 306.057,Z 519.864,A -85,B 0,C 180,E1 -18054.323,E2 -18054.323} C_VEL
LIN {X 0,Y 305.284,Z 533.405,A -85,B 0,C 180,E1 -18055.556,E2 -18055.556} C_VEL
LIN {X 0,Y 304.216,Z 543.172,A -85,B 0,C 180,E1 -18056.19,E2 -18056.19} C_VEL
LIN {X 0,Y 294.562,Z 605.154,A -85,B 0,C 180,E1 -18058.988,E2 -18058.988} C_VEL
LIN {X 0,Y 291.73,Z 618.391,A -85,B 0,C 180,E1 -18059.808,E2 -18059.808} C_VEL
LIN {X 0,Y 288.122,Z 632.396,A -85,B 0,C 180,E1 -18061,E2 -18061} C_VEL
LIN {X 0,Y 284.438,Z 644.805,A -85,B 0,C 180,E1 -18062.401,E2 -18062.401} C_VEL
LIN {X 0,Y 280.971,Z 654.952,A -85,B 0,C 180,E1 -18063.841,E2 -18063.841} C_VEL
LIN {X 0,Y 277.254,Z 665.226,A -85,B 0,C 180,E1 -18065.675,E2 -18065.675} C_VEL
LIN {X 0,Y 273.793,Z 674.123,A -85,B 0,C 180,E1 -18067.675,E2 -18067.675} C_VEL
LIN {X 0,Y 269.96,Z 683.046,A -85,B 0,C 180,E1 -18070.218,E2 -18070.218} C_VEL
LIN {X 0,Y 267.396,Z 688.931,A -85,B 0,C 180,E1 -18072.407,E2 -18072.407} C_VEL
LIN {X 0,Y 265.315,Z 693.632,A -85,B 0,C 180,E1 -18074.639,E2 -18074.639} C_VEL
LIN {X 0,Y 263.688,Z 697.257,A -85,B 0,C 180,E1 -18076.906,E2 -18076.906} C_VEL
LIN {X 0,Y 262.492,Z 699.866,A -85,B 0,C 180,E1 -18079.198,E2 -18079.198} C_VEL
LIN {X 0,Y 261.933,Z 701.061,A -85,B 0,C 180,E1 -18080.736,E2 -18080.736} C_VEL
LIN {X 0,Y 261.515,Z 701.847,A -85,B 0,C 180,E1 -18082.278,E2 -18082.278} C_VEL
LIN {X 0,Y 261.174,Z 702.224,A -85,B 0,C 180,E1 -18084.652,E2 -18084.652} C_VEL
LIN {X 0,Y 261.175,Z 702.161,A -85,B 0,C 180,E1 -18086.915,E2 -18086.915} C_VEL
LIN {X 0,Y 261.164,Z 702.776,A -85,B 0,C 180,E1 -18088.458,E2 -18088.458} C_VEL
LIN {X 0,Y 261.174,Z 702.993,A -85,B 0,C 180,E1 -18090,E2 -18090} C_VEL
LIN {X 0,Y 261.155,Z 702.767,A -85,B 0,C 180,E1 -18091.542,E2 -18091.542} C_VEL
LIN {X 0,Y 261.135,Z 702.145,A -85,B 0,C 180,E1 -18093.086,E2 -18093.086} C_VEL
LIN {X 0,Y 261.132,Z 700.595,A -85,B 0,C 180,E1 -18095.249,E2 -18095.249} C_VEL
LIN {X 0,Y 261.386,Z 697.793,A -85,B 0,C 180,E1 -18097.726,E2 -18097.726} C_VEL
LIN {X 0,Y 261.905,Z 694.11,A -85,B 0,C 180,E1 -18100.045,E2 -18100.045} C_VEL
LIN {X 0,Y 262.683,Z 689.294,A -85,B 0,C 180,E1 -18102.359,E2 -18102.359} C_VEL
LIN {X 0,Y 263.945,Z 683.207,A -85,B 0,C 180,E1 -18104.652,E2 -18104.652} C_VEL
LIN {X 0,Y 265.508,Z 675.618,A -85,B 0,C 180,E1 -18106.928,E2 -18106.928} C_VEL
LIN {X 0,Y 267.047,Z 667.995,A -85,B 0,C 180,E1 -18108.767,E2 -18108.767} C_VEL
LIN {X 0,Y 267.749,Z 664.556,A -85,B 0,C 180,E1 -18109.552,E2 -18109.552} C_VEL
LIN {X 0,Y 271.119,Z 656.065,A -85,B 0,C 180,E1 -18112.078,E2 -18112.078} C_VEL
LIN {X 0,Y 274.699,Z 647.201,A -85,B 0,C 180,E1 -18114.164,E2 -18114.164} C_VEL
LIN {X 0,Y 278.828,Z 636.433,A -85,B 0,C 180,E1 -18116.174,E2 -18116.174} C_VEL
LIN {X 0,Y 283.162,Z 624.448,A -85,B 0,C 180,E1 -18117.935,E2 -18117.935} C_VEL
LIN {X 0,Y 287.569,Z 610.961,A -85,B 0,C 180,E1 -18119.462,E2 -18119.462} C_VEL
LIN {X 0,Y 290.939,Z 599.39,A -85,B 0,C 180,E1 -18120.483,E2 -18120.483} C_VEL
LIN {X 0,Y 294.418,Z 584.963,A -85,B 0,C 180,E1 -18121.478,E2 -18121.478} C_VEL
LIN {X 0,Y 297.33,Z 569.201,A -85,B 0,C 180,E1 -18122.28,E2 -18122.28} C_VEL
LIN {X 0,Y 301.667,Z 538.722,A -85,B 0,C 180,E1 -18123.649,E2 -18123.649} C_VEL
LIN {X 0,Y 302.206,Z 528.821,A -85,B 0,C 180,E1 -18124.415,E2 -18124.415} C_VEL
LIN {X 0,Y 302.413,Z 516.648,A -85,B 0,C 180,E1 -18125.605,E2 -18125.605} C_VEL
LIN {X 0,Y 302.23,Z 508.298,A -85,B 0,C 180,E1 -18126.653,E2 -18126.653} C_VEL
LIN {X 0,Y 300.544,Z 502.555,A -85,B 0,C 180,E1 -18128.247,E2 -18128.247} C_VEL
LIN {X 0,Y 298.865,Z 496.849,A -85,B 0,C 180,E1 -18130.293,E2 -18130.293} C_VEL
LIN {X 0,Y 297.342,Z 492.212,A -85,B 0,C 180,E1 -18133.025,E2 -18133.025} C_VEL
LIN {X 0,Y 296.986,Z 489.947,A -85,B 0,C 180,E1 -18135.098,E2 -18135.098} C_VEL
LIN {X 0,Y 297.241,Z 488.936,A -85,B 0,C 180,E1 -18137.136,E2 -18137.136} C_VEL
LIN {X 0,Y 298.864,Z 488.885,A -85,B 0,C 180,E1 -18140.067,E2 -18140.067} C_VEL
LIN {X 0,Y 301.021,Z 491.192,A -85,B 0,C 180,E1 -18142.446,E2 -18142.446} C_VEL
LIN {X 0,Y 303.4,Z 494.188,A -85,B 0,C 180,E1 -18144.328,E2 -18144.328} C_VEL
LIN {X 0,Y 306.29,Z 498.649,A -85,B 0,C 180,E1 -18146.2,E2 -18146.2} C_VEL
LIN {X 0,Y 306.598,Z 499.277,A -85,B 0,C 180,E1 -18146.392,E2 -18146.392} C_VEL
LIN {X 0,Y 300.207,Z 539.873,A -85,B 0,C 180,E1 -18148.215,E2 -18148.215} C_VEL
LIN {X 0,Y 298.223,Z 553.264,A -85,B 0,C 180,E1 -18148.968,E2 -18148.968} C_VEL
LIN {X 0,Y 295.59,Z 567.112,A -85,B 0,C 180,E1 -18150.046,E2 -18150.046} C_VEL
LIN {X 0,Y 292.259,Z 580.727,A -85,B 0,C 180,E1 -18151.449,E2 -18151.449} C_VEL
LIN {X 0,Y 288.65,Z 592.654,A -85,B 0,C 180,E1 -18153.033,E2 -18153.033} C_VEL
LIN {X 0,Y 285.633,Z 601.559,A -85,B 0,C 180,E1 -18154.495,E2 -18154.495} C_VEL
LIN {X 0,Y 282.427,Z 609.825,A -85,B 0,C 180,E1 -18156.148,E2 -18156.148} C_VEL
LIN {X 0,Y 278.394,Z 619.173,A -85,B 0,C 180,E1 -18158.528,E2 -18158.528} C_VEL
LIN {X 0,Y 275.31,Z 625.564,A -85,B 0,C 180,E1 -18160.618,E2 -18160.618} C_VEL
LIN {X 0,Y 272.366,Z 630.835,A -85,B 0,C 180,E1 -18162.834,E2 -18162.834} C_VEL
LIN {X 0,Y 270.021,Z 634.64,A -85,B 0,C 180,E1 -18164.914,E2 -18164.914} C_VEL
LIN {X 0,Y 268.54,Z 636.682,A -85,B 0,C 180,E1 -18166.377,E2 -18166.377} C_VEL
LIN {X 0,Y 267.177,Z 638.3,A -85,B 0,C 180,E1 -18167.852,E2 -18167.852} C_VEL
LIN {X 0,Y 265.977,Z 639.496,A -85,B 0,C 180,E1 -18169.341,E2 -18169.341} C_VEL
LIN {X 0,Y 265.013,Z 640.237,A -85,B 0,C 180,E1 -18170.844,E2 -18170.844} C_VEL
LIN {X 0,Y 264.232,Z 640.559,A -85,B 0,C 180,E1 -18172.358,E2 -18172.358} C_VEL
LIN {X 0,Y 263.562,Z 640.484,A -85,B 0,C 180,E1 -18173.877,E2 -18173.877} C_VEL
LIN {X 0,Y 262.942,Z 640.002,A -85,B 0,C 180,E1 -18175.401,E2 -18175.401} C_VEL
LIN {X 0,Y 262.447,Z 639.068,A -85,B 0,C 180,E1 -18176.93,E2 -18176.93} C_VEL
LIN {X 0,Y 262.134,Z 637.721,A -85,B 0,C 180,E1 -18178.464,E2 -18178.464} C_VEL
LIN {X 0,Y 261.911,Z 634.88,A -85,B 0,C 180,E1 -18180.769,E2 -18180.769} C_VEL
LIN {X 0,Y 261.904,Z 631.004,A -85,B 0,C 180,E1 -18183.077,E2 -18183.077} C_VEL
LIN {X 0,Y 262.198,Z 625.999,A -85,B 0,C 180,E1 -18185.383,E2 -18185.383} C_VEL
LIN {X 0,Y 262.366,Z 619.713,A -85,B 0,C 180,E1 -18187.697,E2 -18187.697} C_VEL
LIN {X 0,Y 262.866,Z 611.858,A -85,B 0,C 180,E1 -18190.008,E2 -18190.008} C_VEL
LIN {X 0,Y 263.683,Z 602.167,A -85,B 0,C 180,E1 -18192.312,E2 -18192.312} C_VEL
LIN {X 0,Y 264.523,Z 591.092,A -85,B 0,C 180,E1 -18194.423,E2 -18194.423} C_VEL
LIN {X 0,Y 265.393,Z 579.974,A -85,B 0,C 180,E1 -18196.144,E2 -18196.144} C_VEL
LIN {X 0,Y 266.344,Z 567.669,A -85,B 0,C 180,E1 -18197.665,E2 -18197.665} C_VEL
LIN {X 0,Y 267.05,Z 554.742,A -85,B 0,C 180,E1 -18198.929,E2 -18198.929} C_VEL
LIN {X 0,Y 267.845,Z 539.878,A -85,B 0,C 180,E1 -18199.994,E2 -18199.994} C_VEL
LIN {X 0,Y 268.326,Z 524.07,A -85,B 0,C 180,E1 -18200.757,E2 -18200.757} C_VEL
LIN {X 0,Y 270.514,Z 464.924,A -85,B 0,C 180,E1 -18203.176,E2 -18203.176} C_VEL
LIN {X 0,Y 263.199,Z 440.696,A -85,B 0,C 180,E1 -18204.556,E2 -18204.556} C_VEL
LIN {X 0,Y 263.167,Z 440.698,A -85,B 0,C 180,E1 -18208.731,E2 -18208.731} C_VEL
LIN {X 0,Y 263.135,Z 440.684,A -85,B 0,C 180,E1 -18212.288,E2 -18212.288} C_VEL
LIN {X 0,Y 263.187,Z 440.703,A -85,B 0,C 180,E1 -18216.764,E2 -18216.764} C_VEL
LIN {X 0,Y 263.126,Z 440.694,A -85,B 0,C 180,E1 -18221.594,E2 -18221.594} C_VEL
LIN {X 0,Y 263.124,Z 440.71,A -85,B 0,C 180,E1 -18223.984,E2 -18223.984} C_VEL
LIN {X 0,Y 263.126,Z 440.708,A -85,B 0,C 180,E1 -18228.406,E2 -18228.406} C_VEL
LIN {X 0,Y 263.158,Z 440.76,A -85,B 0,C 180,E1 -18230.453,E2 -18230.453} C_VEL
LIN {X 0,Y 266.407,Z 450.991,A -85,B 0,C 180,E1 -18233.573,E2 -18233.573} C_VEL
LIN {X 0,Y 269.545,Z 462.414,A -85,B 0,C 180,E1 -18236.801,E2 -18236.801} C_VEL
LIN {X 0,Y 272.26,Z 474.33,A -85,B 0,C 180,E1 -18239.854,E2 -18239.854} C_VEL
LIN {X 0,Y 274.717,Z 480.817,A -85,B 0,C 180,E1 -18240.375,E2 -18240.375} C_VEL
LIN {X 0,Y 279.381,Z 507.777,A -85,B 0,C 180,E1 -18241.697,E2 -18241.697} C_VEL
LIN {X 0,Y 279.793,Z 512.02,A -85,B 0,C 180,E1 -18241.864,E2 -18241.864} C_VEL
LIN {X 0,Y 277.752,Z 579.239,A -85,B 0,C 180,E1 -18243.565,E2 -18243.565} C_VEL
LIN {X 0,Y 277.042,Z 592.955,A -85,B 0,C 180,E1 -18244.049,E2 -18244.049} C_VEL
LIN {X 0,Y 275.911,Z 605.11,A -85,B 0,C 180,E1 -18244.744,E2 -18244.744} C_VEL
LIN {X 0,Y 274.522,Z 618.032,A -85,B 0,C 180,E1 -18245.819,E2 -18245.819} C_VEL
LIN {X 0,Y 272.812,Z 629.448,A -85,B 0,C 180,E1 -18247.068,E2 -18247.068} C_VEL
LIN {X 0,Y 270.838,Z 640.864,A -85,B 0,C 180,E1 -18248.698,E2 -18248.698} C_VEL
LIN {X 0,Y 269.002,Z 651.036,A -85,B 0,C 180,E1 -18250.542,E2 -18250.542} C_VEL
LIN {X 0,Y 267.238,Z 659.283,A -85,B 0,C 180,E1 -18252.396,E2 -18252.396} C_VEL
LIN {X 0,Y 265.37,Z 667.323,A -85,B 0,C 180,E1 -18254.643,E2 -18254.643} C_VEL
LIN {X 0,Y 264.025,Z 673.784,A -85,B 0,C 180,E1 -18256.923,E2 -18256.923} C_VEL
LIN {X 0,Y 262.873,Z 678.922,A -85,B 0,C 180,E1 -18259.214,E2 -18259.214} C_VEL
LIN {X 0,Y 262.109,Z 682.896,A -85,B 0,C 180,E1 -18261.519,E2 -18261.519} C_VEL
LIN {X 0,Y 261.592,Z 685.824,A -85,B 0,C 180,E1 -18263.831,E2 -18263.831} C_VEL
LIN {X 0,Y 261.381,Z 687.242,A -85,B 0,C 180,E1 -18265.373,E2 -18265.373} C_VEL
LIN {X 0,Y 261.244,Z 688.236,A -85,B 0,C 180,E1 -18266.916,E2 -18266.916} C_VEL
LIN {X 0,Y 261.158,Z 688.849,A -85,B 0,C 180,E1 -18268.458,E2 -18268.458} C_VEL
LIN {X 0,Y 261.124,Z 689.081,A -85,B 0,C 180,E1 -18270,E2 -18270} C_VEL
LIN {X 0,Y 261.158,Z 688.885,A -85,B 0,C 180,E1 -18271.542,E2 -18271.542} C_VEL
LIN {X 0,Y 261.243,Z 688.297,A -85,B 0,C 180,E1 -18273.084,E2 -18273.084} C_VEL
LIN {X 0,Y 261.381,Z 687.327,A -85,B 0,C 180,E1 -18274.627,E2 -18274.627} C_VEL
LIN {X 0,Y 261.63,Z 685.782,A -85,B 0,C 180,E1 -18276.325,E2 -18276.325} C_VEL
LIN {X 0,Y 262.288,Z 681.872,A -85,B 0,C 180,E1 -18279.252,E2 -18279.252} C_VEL
LIN {X 0,Y 263.197,Z 677.589,A -85,B 0,C 180,E1 -18281.553,E2 -18281.553} C_VEL
LIN {X 0,Y 264.439,Z 672.114,A -85,B 0,C 180,E1 -18283.839,E2 -18283.839} C_VEL
LIN {X 0,Y 265.922,Z 665.246,A -85,B 0,C 180,E1 -18286.111,E2 -18286.111} C_VEL
LIN {X 0,Y 267.886,Z 656.649,A -85,B 0,C 180,E1 -18288.35,E2 -18288.35} C_VEL
LIN {X 0,Y 269.653,Z 647.682,A -85,B 0,C 180,E1 -18290.235,E2 -18290.235} C_VEL
LIN {X 0,Y 271.359,Z 638.13,A -85,B 0,C 180,E1 -18291.858,E2 -18291.858} C_VEL
LIN {X 0,Y 273.181,Z 627.369,A -85,B 0,C 180,E1 -18293.3,E2 -18293.3} C_VEL
LIN {X 0,Y 274.841,Z 615.402,A -85,B 0,C 180,E1 -18294.553,E2 -18294.553} C_VEL
LIN {X 0,Y 276.272,Z 602.771,A -85,B 0,C 180,E1 -18295.523,E2 -18295.523} C_VEL
LIN {X 0,Y 277.166,Z 590.335,A -85,B 0,C 180,E1 -18296.191,E2 -18296.191} C_VEL
LIN {X 0,Y 277.936,Z 574.699,A -85,B 0,C 180,E1 -18296.669,E2 -18296.669} C_VEL
LIN {X 0,Y 279.854,Z 510.643,A -85,B 0,C 180,E1 -18298.293,E2 -18298.293} C_VEL
LIN {X 0,Y 275.407,Z 484.522,A -85,B 0,C 180,E1 -18299.561,E2 -18299.561} C_VEL
LIN {X 0,Y 274.261,Z 479.386,A -85,B 0,C 180,E1 -18299.849,E2 -18299.849} C_VEL
LIN {X 0,Y 272.306,Z 474.288,A -85,B 0,C 180,E1 -18300.283,E2 -18300.283} C_VEL
LIN {X 0,Y 269.683,Z 462.987,A -85,B 0,C 180,E1 -18303.18,E2 -18303.18} C_VEL
LIN {X 0,Y 266.543,Z 451.342,A -85,B 0,C 180,E1 -18306.466,E2 -18306.466} C_VEL
LIN {X 0,Y 263.155,Z 440.699,A -85,B 0,C 180,E1 -18309.7,E2 -18309.7} C_VEL
LIN {X 0,Y 263.135,Z 440.698,A -85,B 0,C 180,E1 -18313.982,E2 -18313.982} C_VEL
LIN {X 0,Y 263.127,Z 440.695,A -85,B 0,C 180,E1 -18318.406,E2 -18318.406} C_VEL
LIN {X 0,Y 263.187,Z 440.68,A -85,B 0,C 180,E1 -18323.236,E2 -18323.236} C_VEL
LIN {X 0,Y 263.144,Z 440.696,A -85,B 0,C 180,E1 -18325.346,E2 -18325.346} C_VEL
LIN {X 0,Y 262.95,Z 441.363,A -85,B 0,C 180,E1 -18326.178,E2 -18326.178} C_VEL
LIN {X 0,Y 262.273,Z 443.534,A -85,B 0,C 180,E1 -18327.132,E2 -18327.132} C_VEL
LIN {X 0,Y 260.994,Z 447.905,A -85,B 0,C 180,E1 -18328.32,E2 -18328.32} C_VEL
LIN {X 0,Y 259.623,Z 455.082,A -85,B 0,C 180,E1 -18329.913,E2 -18329.913} C_VEL
LIN {X 0,Y 259.871,Z 459.167,A -85,B 0,C 180,E1 -18330.894,E2 -18330.894} C_VEL
LIN {X 0,Y 261.356,Z 466.97,A -85,B 0,C 180,E1 -18332.797,E2 -18332.797} C_VEL
LIN {X 0,Y 260.624,Z 475.275,A -85,B 0,C 180,E1 -18334.674,E2 -18334.674} C_VEL
LIN {X 0,Y 262.958,Z 499.892,A -85,B 0,C 180,E1 -18335.857,E2 -18335.857} C_VEL
LIN {X 0,Y 263.808,Z 507.877,A -85,B 0,C 180,E1 -18336.237,E2 -18336.237} C_VEL
LIN {X 0,Y 260.625,Z 586.91,A -85,B 0,C 180,E1 -18339.633,E2 -18339.633} C_VEL
LIN {X 0,Y 259.909,Z 601.104,A -85,B 0,C 180,E1 -18340.553,E2 -18340.553} C_VEL
LIN {X 0,Y 258.964,Z 614.5,A -85,B 0,C 180,E1 -18341.752,E2 -18341.752} C_VEL
LIN {X 0,Y 257.983,Z 626.785,A -85,B 0,C 180,E1 -18343.175,E2 -18343.175} C_VEL
LIN {X 0,Y 257.131,Z 637.58,A -85,B 0,C 180,E1 -18344.747,E2 -18344.747} C_VEL
LIN {X 0,Y 256.256,Z 647.597,A -85,B 0,C 180,E1 -18346.519,E2 -18346.519} C_VEL
LIN {X 0,Y 255.513,Z 656.767,A -85,B 0,C 180,E1 -18348.497,E2 -18348.497} C_VEL
LIN {X 0,Y 254.835,Z 665.694,A -85,B 0,C 180,E1 -18350.876,E2 -18350.876} C_VEL
LIN {X 0,Y 254.377,Z 672.834,A -85,B 0,C 180,E1 -18353.257,E2 -18353.257} C_VEL
LIN {X 0,Y 254.15,Z 679.375,A -85,B 0,C 180,E1 -18356.036,E2 -18356.036} C_VEL
LIN {X 0,Y 254.069,Z 683.609,A -85,B 0,C 180,E1 -18358.415,E2 -18358.415} C_VEL
LIN {X 0,Y 254.046,Z 685.775,A -85,B 0,C 180,E1 -18360,E2 -18360} C_VEL
LIN {X 0,Y 254.107,Z 687.511,A -85,B 0,C 180,E1 -18361.585,E2 -18361.585} C_VEL
LIN {X 0,Y 254.189,Z 688.79,A -85,B 0,C 180,E1 -18363.17,E2 -18363.17} C_VEL
LIN {X 0,Y 254.754,Z 690.045,A -85,B 0,C 180,E1 -18366.335,E2 -18366.335} C_VEL
LIN {X 0,Y 255.247,Z 690.071,A -85,B 0,C 180,E1 -18367.913,E2 -18367.913} C_VEL
LIN {X 0,Y 255.846,Z 689.644,A -85,B 0,C 180,E1 -18369.487,E2 -18369.487} C_VEL
LIN {X 0,Y 257.692,Z 687.596,A -85,B 0,C 180,E1 -18372.602,E2 -18372.602} C_VEL
LIN {X 0,Y 259.399,Z 684.95,A -85,B 0,C 180,E1 -18374.915,E2 -18374.915} C_VEL
LIN {X 0,Y 261.718,Z 681.269,A -85,B 0,C 180,E1 -18377.181,E2 -18377.181} C_VEL
LIN {X 0,Y 264.403,Z 676.538,A -85,B 0,C 180,E1 -18379.406,E2 -18379.406} C_VEL
LIN {X 0,Y 267.506,Z 670.546,A -85,B 0,C 180,E1 -18381.581,E2 -18381.581} C_VEL
LIN {X 0,Y 271.693,Z 661.862,A -85,B 0,C 180,E1 -18384.042,E2 -18384.042} C_VEL
LIN {X 0,Y 275.689,Z 652.528,A -85,B 0,C 180,E1 -18386.088,E2 -18386.088} C_VEL
LIN {X 0,Y 279.69,Z 642.302,A -85,B 0,C 180,E1 -18387.874,E2 -18387.874} C_VEL
LIN {X 0,Y 283.496,Z 631.15,A -85,B 0,C 180,E1 -18389.428,E2 -18389.428} C_VEL
